KUKA KRL data list: CNC3.dat

&ACCESS RV
DEFDAT CNC3 Public
DECL GLOBAL FRAME gfCNCPoint3[30000]


gfCNCPoint3[1] = {X 137.7105, Y 20.4366, Z -3.8333, A 0.000, B 0.000, C 0.000 }
gfCNCPoint3[2] = {X 137.0001, Y 21.1821, Z -3.8333, A 0.000, B 0.000, C 0.000 }
gfCNCPoint3[3] = {X 136.1491, Y 21.7619, Z -3.8333, A 0.000, B 0.000, C 0.000 }
gfCNCPoint3[4] = {X 135.4282, Y 22.0767, Z -3.8333, A 0.000, B 0.000, C 0.000 }
gfCNCPoint3[5] = {X 134.6660, Y 22.2715, Z -3.8333, A 0.000, B 0.000, C 0.000 }
gfCNCPoint3[6] = {X 133.8824, Y 22.3414, Z -3.8333, A 0.000, B 0.000, C 0.000 }
gfCNCPoint3[7] = {X 133.2006, Y 22.3415, Z -3.8333, A 0.000, B 0.000, C 0.000 }
gfCNCPoint3[8] = {X 132.2486, Y 22.2478, Z -3.8333, A 0.000, B 0.000, C 0.000 }
gfCNCPoint3[9] = {X 131.3331, Y 21.9701, Z -3.8333, A 0.000, B 0.000, C 0.000 }
gfCNCPoint3[10] = {X 130.4895, Y 21.5191, Z -3.8333, A 0.000, B 0.000, C 0.000 }
gfCNCPoint3[11] = {X 129.7500, Y 20.9122, Z -3.8333, A 0.000, B 0.000, C 0.000 }
gfCNCPoint3[12] = {X 129.1431, Y 20.1727, Z -3.8333, A 0.000, B 0.000, C 0.000 }
gfCNCPoint3[13] = {X 128.6921, Y 19.3290, Z -3.8333, A 0.000, B 0.000, C 0.000 }
gfCNCPoint3[14] = {X 128.4144, Y 18.4136, Z -3.8333, A 0.000, B 0.000, C 0.000 }
gfCNCPoint3[15] = {X 128.3206, Y 17.4615, Z -3.8333, A 0.000, B 0.000, C 0.000 }
gfCNCPoint3[16] = {X 128.3206, Y 10.4835, Z -3.8333, A 0.000, B 0.000, C 0.000 }
gfCNCPoint3[17] = {X 128.3317, Y 10.1548, Z -3.8333, A 0.000, B 0.000, C 0.000 }
gfCNCPoint3[18] = {X 128.3649, Y 9.8276, Z -3.8333, A 0.000, B 0.000, C 0.000 }
gfCNCPoint3[19] = {X 128.6078, Y 8.8341, Z -3.8333, A 0.000, B 0.000, C 0.000 }
gfCNCPoint3[20] = {X 129.0525, Y 7.9131, Z -3.8333, A 0.000, B 0.000, C 0.000 }
gfCNCPoint3[21] = {X 129.6793, Y 7.1050, Z -3.8333, A 0.000, B 0.000, C 0.000 }
gfCNCPoint3[22] = {X 130.0256, Y 7.4373, Z -3.8333, A 0.000, B 0.000, C 0.000 }
gfCNCPoint3[23] = {X 130.6996, Y 6.8634, Z -3.8333, A 0.000, B 0.000, C 0.000 }
gfCNCPoint3[24] = {X 131.4749, Y 6.4361, Z -3.8333, A 0.000, B 0.000, C 0.000 }
gfCNCPoint3[25] = {X 132.3199, Y 6.1726, Z -3.8333, A 0.000, B 0.000, C 0.000 }
gfCNCPoint3[26] = {X 133.2007, Y 6.0835, Z -3.8333, A 0.000, B 0.000, C 0.000 }
gfCNCPoint3[27] = {X 133.8874, Y 6.0837, Z -3.8333, A 0.000, B 0.000, C 0.000 }
gfCNCPoint3[28] = {X 134.7189, Y 6.1717, Z -3.8333, A 0.000, B 0.000, C 0.000 }
gfCNCPoint3[29] = {X 135.5188, Y 6.4154, Z -3.8333, A 0.000, B 0.000, C 0.000 }
gfCNCPoint3[30] = {X 136.2581, Y 6.8060, Z -3.8333, A 0.000, B 0.000, C 0.000 }
gfCNCPoint3[31] = {X 136.9101, Y 7.3294, Z -3.8333, A 0.000, B 0.000, C 0.000 }
gfCNCPoint3[32] = {X 137.4514, Y 7.9667, Z -3.8333, A 0.000, B 0.000, C 0.000 }
gfCNCPoint3[33] = {X 155.0713, Y 7.9667, Z -3.8333, A 0.000, B 0.000, C 0.000 }
gfCNCPoint3[34] = {X 155.6191, Y 7.3231, Z -3.8333, A 0.000, B 0.000, C 0.000 }
gfCNCPoint3[35] = {X 156.2798, Y 6.7961, Z -3.8333, A 0.000, B 0.000, C 0.000 }
gfCNCPoint3[36] = {X 157.0291, Y 6.4051, Z -3.8333, A 0.000, B 0.000, C 0.000 }
gfCNCPoint3[37] = {X 157.8393, Y 6.1647, Z -3.8333, A 0.000, B 0.000, C 0.000 }
gfCNCPoint3[38] = {X 158.6806, Y 6.0835, Z -3.8333, A 0.000, B 0.000, C 0.000 }
gfCNCPoint3[39] = {X 159.3791, Y 6.0839, Z -3.8333, A 0.000, B 0.000, C 0.000 }
gfCNCPoint3[40] = {X 160.3488, Y 6.2050, Z -3.8333, A 0.000, B 0.000, C 0.000 }
gfCNCPoint3[41] = {X 161.2678, Y 6.5371, Z -3.8333, A 0.000, B 0.000, C 0.000 }
gfCNCPoint3[42] = {X 162.0908, Y 7.0639, Z -3.8333, A 0.000, B 0.000, C 0.000 }
gfCNCPoint3[43] = {X 162.7773, Y 7.7593, Z -3.8333, A 0.000, B 0.000, C 0.000 }
gfCNCPoint3[44] = {X 163.2934, Y 8.5891, Z -3.8333, A 0.000, B 0.000, C 0.000 }
gfCNCPoint3[45] = {X 163.6136, Y 9.5124, Z -3.8333, A 0.000, B 0.000, C 0.000 }
gfCNCPoint3[46] = {X 163.7221, Y 10.4835, Z -3.8333, A 0.000, B 0.000, C 0.000 }
gfCNCPoint3[47] = {X 163.7221, Y 17.4615, Z -3.8333, A 0.000, B 0.000, C 0.000 }
gfCNCPoint3[48] = {X 163.6118, Y 18.4406, Z -3.8333, A 0.000, B 0.000, C 0.000 }
gfCNCPoint3[49] = {X 163.2863, Y 19.3706, Z -3.8333, A 0.000, B 0.000, C 0.000 }
gfCNCPoint3[50] = {X 162.7621, Y 20.2049, Z -3.8333, A 0.000, B 0.000, C 0.000 }
gfCNCPoint3[51] = {X 162.0654, Y 20.9016, Z -3.8333, A 0.000, B 0.000, C 0.000 }
gfCNCPoint3[52] = {X 161.2312, Y 21.4258, Z -3.8333, A 0.000, B 0.000, C 0.000 }
gfCNCPoint3[53] = {X 160.3012, Y 21.7512, Z -3.8333, A 0.000, B 0.000, C 0.000 }
gfCNCPoint3[54] = {X 159.3221, Y 21.8615, Z -3.8333, A 0.000, B 0.000, C 0.000 }
gfCNCPoint3[55] = {X 158.6788, Y 21.8615, Z -3.8333, A 0.000, B 0.000, C 0.000 }
gfCNCPoint3[56] = {X 157.8334, Y 21.7764, Z -3.8333, A 0.000, B 0.000, C 0.000 }
gfCNCPoint3[57] = {X 157.0197, Y 21.5317, Z -3.8333, A 0.000, B 0.000, C 0.000 }
gfCNCPoint3[58] = {X 156.2677, Y 21.1363, Z -3.8333, A 0.000, B 0.000, C 0.000 }
gfCNCPoint3[59] = {X 155.6048, Y 20.6048, Z -3.8333, A 0.000, B 0.000, C 0.000 }
gfCNCPoint3[60] = {X 155.0554, Y 19.9566, Z -3.8333, A 0.000, B 0.000, C 0.000 }
gfCNCPoint3[61] = {X 152.3562, Y 19.9578, Z -3.8333, A 0.000, B 0.000, C 0.000 }
gfCNCPoint3[62] = {X 152.3548, Y 40.8428, Z -3.8333, A 0.000, B 0.000, C 0.000 }
gfCNCPoint3[63] = {X 152.8075, Y 41.3308, Z -3.8333, A 0.000, B 0.000, C 0.000 }
gfCNCPoint3[64] = {X 152.8997, Y 41.4410, Z -3.8333, A 0.000, B 0.000, C 0.000 }
gfCNCPoint3[65] = {X 153.4341, Y 42.2814, Z -3.8333, A 0.000, B 0.000, C 0.000 }
gfCNCPoint3[66] = {X 153.7674, Y 43.2198, Z -3.8333, A 0.000, B 0.000, C 0.000 }
gfCNCPoint3[67] = {X 153.8831, Y 44.2089, Z -3.8333, A 0.000, B 0.000, C 0.000 }
gfCNCPoint3[68] = {X 153.8829, Y 45.0423, Z -3.8333, A 0.000, B 0.000, C 0.000 }
gfCNCPoint3[69] = {X 153.7646, Y 46.0144, Z -3.8333, A 0.000, B 0.000, C 0.000 }
gfCNCPoint3[70] = {X 153.4342, Y 46.9363, Z -3.8333, A 0.000, B 0.000, C 0.000 }
gfCNCPoint3[71] = {X 152.9080, Y 47.7622, Z -3.8333, A 0.000, B 0.000, C 0.000 }
gfCNCPoint3[72] = {X 152.2123, Y 48.4513, Z -3.8333, A 0.000, B 0.000, C 0.000 }
gfCNCPoint3[73] = {X 151.3813, Y 48.9695, Z -3.8333, A 0.000, B 0.000, C 0.000 }
gfCNCPoint3[74] = {X 150.4563, Y 49.2910, Z -3.8333, A 0.000, B 0.000, C 0.000 }
gfCNCPoint3[75] = {X 149.4831, Y 49.4000, Z -3.8333, A 0.000, B 0.000, C 0.000 }
gfCNCPoint3[76] = {X 143.0396, Y 49.4000, Z -3.8333, A 0.000, B 0.000, C 0.000 }
gfCNCPoint3[77] = {X 142.0605, Y 49.2897, Z -3.8333, A 0.000, B 0.000, C 0.000 }
gfCNCPoint3[78] = {X 141.1305, Y 48.9643, Z -3.8333, A 0.000, B 0.000, C 0.000 }
gfCNCPoint3[79] = {X 140.2963, Y 48.4400, Z -3.8333, A 0.000, B 0.000, C 0.000 }
gfCNCPoint3[80] = {X 139.5996, Y 47.7433, Z -3.8333, A 0.000, B 0.000, C 0.000 }
gfCNCPoint3[81] = {X 139.0754, Y 46.9091, Z -3.8333, A 0.000, B 0.000, C 0.000 }
gfCNCPoint3[82] = {X 138.7499, Y 45.9791, Z -3.8333, A 0.000, B 0.000, C 0.000 }
gfCNCPoint3[83] = {X 138.6396, Y 45.0000, Z -3.8333, A 0.000, B 0.000, C 0.000 }
gfCNCPoint3[84] = {X 138.6400, Y 44.1483, Z -3.8333, A 0.000, B 0.000, C 0.000 }
gfCNCPoint3[85] = {X 138.7505, Y 43.2275, Z -3.8333, A 0.000, B 0.000, C 0.000 }
gfCNCPoint3[86] = {X 139.0514, Y 42.3503, Z -3.8333, A 0.000, B 0.000, C 0.000 }
gfCNCPoint3[87] = {X 139.5295, Y 41.5556, Z -3.8333, A 0.000, B 0.000, C 0.000 }
gfCNCPoint3[88] = {X 140.1636, Y 40.8789, Z -3.8333, A 0.000, B 0.000, C 0.000 }
gfCNCPoint3[89] = {X 140.1636, Y 19.9572, Z -3.8333, A 0.000, B 0.000, C 0.000 }
gfCNCPoint3[90] = {X 137.4665, Y 19.9566, Z -3.8333, A 0.000, B 0.000, C 0.000 }
gfCNCPoint3[91] = {X 136.9188, Y 20.6072, Z -3.8333, A 0.000, B 0.000, C 0.000 }
gfCNCPoint3[92] = {X 136.2562, Y 21.1403, Z -3.8333, A 0.000, B 0.000, C 0.000 }
gfCNCPoint3[93] = {X 135.5034, Y 21.5359, Z -3.8333, A 0.000, B 0.000, C 0.000 }
gfCNCPoint3[94] = {X 134.6886, Y 21.7794, Z -3.8333, A 0.000, B 0.000, C 0.000 }
gfCNCPoint3[95] = {X 133.8422, Y 21.8615, Z -3.8333, A 0.000, B 0.000, C 0.000 }
gfCNCPoint3[96] = {X 133.2006, Y 21.8615, Z -3.8333, A 0.000, B 0.000, C 0.000 }
gfCNCPoint3[97] = {X 132.2215, Y 21.7512, Z -3.8333, A 0.000, B 0.000, C 0.000 }
gfCNCPoint3[98] = {X 131.2916, Y 21.4258, Z -3.8333, A 0.000, B 0.000, C 0.000 }
gfCNCPoint3[99] = {X 130.4573, Y 20.9016, Z -3.8333, A 0.000, B 0.000, C 0.000 }
gfCNCPoint3[100] = {X 129.7606, Y 20.2049, Z -3.8333, A 0.000, B 0.000, C 0.000 }
gfCNCPoint3[101] = {X 129.2364, Y 19.3706, Z -3.8333, A 0.000, B 0.000, C 0.000 }
gfCNCPoint3[102] = {X 128.9110, Y 18.4406, Z -3.8333, A 0.000, B 0.000, C 0.000 }
gfCNCPoint3[103] = {X 128.8006, Y 17.4615, Z -3.8333, A 0.000, B 0.000, C 0.000 }
gfCNCPoint3[104] = {X 128.8006, Y 10.4835, Z -3.8333, A 0.000, B 0.000, C 0.000 }
gfCNCPoint3[105] = {X 128.8808, Y 9.6475, Z -3.8333, A 0.000, B 0.000, C 0.000 }
gfCNCPoint3[106] = {X 129.1184, Y 8.8419, Z -3.8333, A 0.000, B 0.000, C 0.000 }
gfCNCPoint3[107] = {X 129.5047, Y 8.0961, Z -3.8333, A 0.000, B 0.000, C 0.000 }
gfCNCPoint3[108] = {X 130.0256, Y 7.4373, Z -3.8333, A 0.000, B 0.000, C 0.000 }
gfCNCPoint3[109] = {X 129.6793, Y 7.1050, Z -3.8333, A 0.000, B 0.000, C 0.000 }
gfCNCPoint3[110] = {X 102.4337, Y 7.1050, Z -3.8333, A 0.000, B 0.000, C 0.000 }
gfCNCPoint3[111] = {X 102.4337, Y 11.9050, Z -3.8333, A 0.000, B 0.000, C 0.000 }
gfCNCPoint3[112] = {X 101.3242, Y 11.9050, Z -3.8333, A 0.000, B 0.000, C 0.000 }
gfCNCPoint3[113] = {X 101.3283, Y 12.0459, Z -3.8333, A 0.000, B 0.000, C 0.000 }
gfCNCPoint3[114] = {X 101.3297, Y 12.1868, Z -3.8333, A 0.000, B 0.000, C 0.000 }
gfCNCPoint3[115] = {X 101.3293, Y 13.0462, Z -3.8333, A 0.000, B 0.000, C 0.000 }
gfCNCPoint3[116] = {X 101.2274, Y 14.1939, Z -3.8333, A 0.000, B 0.000, C 0.000 }
gfCNCPoint3[117] = {X 100.9457, Y 15.3111, Z -3.8333, A 0.000, B 0.000, C 0.000 }
gfCNCPoint3[118] = {X 101.0393, Y 15.5442, Z -3.8333, A 0.000, B 0.000, C 0.000 }
gfCNCPoint3[119] = {X 101.8684, Y 17.5994, Z -3.8333, A 0.000, B 0.000, C 0.000 }
gfCNCPoint3[120] = {X 102.8003, Y 15.2755, Z -3.8333, A 0.000, B 0.000, C 0.000 }
gfCNCPoint3[121] = {X 102.5264, Y 14.1695, Z -3.8333, A 0.000, B 0.000, C 0.000 }
gfCNCPoint3[122] = {X 102.4285, Y 13.0344, Z -3.8333, A 0.000, B 0.000, C 0.000 }
gfCNCPoint3[123] = {X 102.4283, Y 12.1868, Z -3.8333, A 0.000, B 0.000, C 0.000 }
gfCNCPoint3[124] = {X 102.4296, Y 12.0459, Z -3.8333, A 0.000, B 0.000, C 0.000 }
gfCNCPoint3[125] = {X 102.4337, Y 11.9050, Z -3.8333, A 0.000, B 0.000, C 0.000 }
gfCNCPoint3[126] = {X 102.4337, Y 9.5050, Z -3.8333, A 0.000, B 0.000, C 0.000 }
gfCNCPoint3[127] = {X 98.1267, Y 9.5050, Z -3.8333, A 0.000, B 0.000, C 0.000 }
gfCNCPoint3[128] = {X 98.5429, Y 10.2829, Z -3.8333, A 0.000, B 0.000, C 0.000 }
gfCNCPoint3[129] = {X 98.8123, Y 11.1230, Z -3.8333, A 0.000, B 0.000, C 0.000 }
gfCNCPoint3[130] = {X 98.9260, Y 11.9979, Z -3.8333, A 0.000, B 0.000, C 0.000 }
gfCNCPoint3[131] = {X 98.9288, Y 12.0923, Z -3.8333, A 0.000, B 0.000, C 0.000 }
gfCNCPoint3[132] = {X 98.9297, Y 12.1868, Z -3.8333, A 0.000, B 0.000, C 0.000 }
gfCNCPoint3[133] = {X 98.9294, Y 13.0237, Z -3.8333, A 0.000, B 0.000, C 0.000 }
gfCNCPoint3[134] = {X 98.8589, Y 13.8059, Z -3.8333, A 0.000, B 0.000, C 0.000 }
gfCNCPoint3[135] = {X 98.6639, Y 14.5666, Z -3.8333, A 0.000, B 0.000, C 0.000 }
gfCNCPoint3[136] = {X 98.3493, Y 15.2862, Z -3.8333, A 0.000, B 0.000, C 0.000 }
gfCNCPoint3[137] = {X 98.8129, Y 16.4405, Z -3.8333, A 0.000, B 0.000, C 0.000 }
gfCNCPoint3[138] = {X 101.8752, Y 24.0312, Z -3.8333, A 0.000, B 0.000, C 0.000 }
gfCNCPoint3[139] = {X 105.3933, Y 15.2574, Z -3.8333, A 0.000, B 0.000, C 0.000 }
gfCNCPoint3[140] = {X 105.0870, Y 14.5458, Z -3.8333, A 0.000, B 0.000, C 0.000 }
gfCNCPoint3[141] = {X 104.8971, Y 13.7947, Z -3.8333, A 0.000, B 0.000, C 0.000 }
gfCNCPoint3[142] = {X 104.8285, Y 13.0231, Z -3.8333, A 0.000, B 0.000, C 0.000 }
gfCNCPoint3[143] = {X 104.8283, Y 12.1868, Z -3.8333, A 0.000, B 0.000, C 0.000 }
gfCNCPoint3[144] = {X 104.8292, Y 12.0923, Z -3.8333, A 0.000, B 0.000, C 0.000 }
gfCNCPoint3[145] = {X 104.8319, Y 11.9979, Z -3.8333, A 0.000, B 0.000, C 0.000 }
gfCNCPoint3[146] = {X 104.9456, Y 11.1230, Z -3.8333, A 0.000, B 0.000, C 0.000 }
gfCNCPoint3[147] = {X 105.2150, Y 10.2829, Z -3.8333, A 0.000, B 0.000, C 0.000 }
gfCNCPoint3[148] = {X 105.6312, Y 9.5050, Z -3.8333, A 0.000, B 0.000, C 0.000 }
gfCNCPoint3[149] = {X 102.4337, Y 9.5050, Z -3.8333, A 0.000, B 0.000, C 0.000 }
gfCNCPoint3[150] = {X 102.4337, Y 7.1050, Z -3.8333, A 0.000, B 0.000, C 0.000 }
gfCNCPoint3[151] = {X 64.8350, Y 7.1050, Z -3.8333, A 0.000, B 0.000, C 0.000 }
gfCNCPoint3[152] = {X 65.5946, Y 8.0242, Z -3.8333, A 0.000, B 0.000, C 0.000 }
gfCNCPoint3[153] = {X 66.1941, Y 9.0550, Z -3.8333, A 0.000, B 0.000, C 0.000 }
gfCNCPoint3[154] = {X 66.6172, Y 10.1699, Z -3.8333, A 0.000, B 0.000, C 0.000 }
gfCNCPoint3[155] = {X 66.8305, Y 11.1683, Z -3.8333, A 0.000, B 0.000, C 0.000 }
gfCNCPoint3[156] = {X 66.9021, Y 12.1868, Z -3.8333, A 0.000, B 0.000, C 0.000 }
gfCNCPoint3[157] = {X 66.9018, Y 13.0462, Z -3.8333, A 0.000, B 0.000, C 0.000 }
gfCNCPoint3[158] = {X 66.7772, Y 14.3210, Z -3.8333, A 0.000, B 0.000, C 0.000 }
gfCNCPoint3[159] = {X 66.4310, Y 15.5543, Z -3.8333, A 0.000, B 0.000, C 0.000 }
gfCNCPoint3[160] = {X 74.9112, Y 38.2391, Z -3.8333, A 0.000, B 0.000, C 0.000 }
gfCNCPoint3[161] = {X 75.8036, Y 38.9739, Z -3.8333, A 0.000, B 0.000, C 0.000 }
gfCNCPoint3[162] = {X 76.5684, Y 39.8407, Z -3.8333, A 0.000, B 0.000, C 0.000 }
gfCNCPoint3[163] = {X 77.1864, Y 40.8176, Z -3.8333, A 0.000, B 0.000, C 0.000 }
gfCNCPoint3[164] = {X 77.6419, Y 41.8800, Z -3.8333, A 0.000, B 0.000, C 0.000 }
gfCNCPoint3[165] = {X 77.9236, Y 43.0011, Z -3.8333, A 0.000, B 0.000, C 0.000 }
gfCNCPoint3[166] = {X 78.0243, Y 44.1527, Z -3.8333, A 0.000, B 0.000, C 0.000 }
gfCNCPoint3[167] = {X 78.0245, Y 45.0000, Z -3.8333, A 0.000, B 0.000, C 0.000 }
gfCNCPoint3[168] = {X 77.9139, Y 46.2642, Z -3.8333, A 0.000, B 0.000, C 0.000 }
gfCNCPoint3[169] = {X 77.5854, Y 47.4899, Z -3.8333, A 0.000, B 0.000, C 0.000 }
gfCNCPoint3[170] = {X 77.0491, Y 48.6400, Z -3.8333, A 0.000, B 0.000, C 0.000 }
gfCNCPoint3[171] = {X 76.3213, Y 49.6795, Z -3.8333, A 0.000, B 0.000, C 0.000 }
gfCNCPoint3[172] = {X 75.4240, Y 50.5768, Z -3.8333, A 0.000, B 0.000, C 0.000 }
gfCNCPoint3[173] = {X 74.3845, Y 51.3047, Z -3.8333, A 0.000, B 0.000, C 0.000 }
gfCNCPoint3[174] = {X 73.2344, Y 51.8410, Z -3.8333, A 0.000, B 0.000, C 0.000 }
gfCNCPoint3[175] = {X 72.0086, Y 52.1694, Z -3.8333, A 0.000, B 0.000, C 0.000 }
gfCNCPoint3[176] = {X 70.7445, Y 52.2800, Z -3.8333, A 0.000, B 0.000, C 0.000 }
gfCNCPoint3[177] = {X 64.1851, Y 52.2800, Z -3.8333, A 0.000, B 0.000, C 0.000 }
gfCNCPoint3[178] = {X 62.9397, Y 52.1727, Z -3.8333, A 0.000, B 0.000, C 0.000 }
gfCNCPoint3[179] = {X 61.7311, Y 51.8539, Z -3.8333, A 0.000, B 0.000, C 0.000 }
gfCNCPoint3[180] = {X 60.5947, Y 51.3330, Z -3.8333, A 0.000, B 0.000, C 0.000 }
gfCNCPoint3[181] = {X 59.5643, Y 50.6255, Z -3.8333, A 0.000, B 0.000, C 0.000 }
gfCNCPoint3[182] = {X 58.6700, Y 49.7521, Z -3.8333, A 0.000, B 0.000, C 0.000 }
gfCNCPoint3[183] = {X 57.9384, Y 48.7385, Z -3.8333, A 0.000, B 0.000, C 0.000 }
gfCNCPoint3[184] = {X 57.3706, Y 47.5614, Z -3.8333, A 0.000, B 0.000, C 0.000 }
gfCNCPoint3[185] = {X 57.0224, Y 46.3017, Z -3.8333, A 0.000, B 0.000, C 0.000 }
gfCNCPoint3[186] = {X 56.9051, Y 45.0000, Z -3.8333, A 0.000, B 0.000, C 0.000 }
gfCNCPoint3[187] = {X 56.9051, Y 44.2047, Z -3.8333, A 0.000, B 0.000, C 0.000 }
gfCNCPoint3[188] = {X 56.9286, Y 43.6251, Z -3.8333, A 0.000, B 0.000, C 0.000 }
gfCNCPoint3[189] = {X 56.9981, Y 43.0492, Z -3.8333, A 0.000, B 0.000, C 0.000 }
gfCNCPoint3[190] = {X 54.7600, Y 43.0492, Z -3.8333, A 0.000, B 0.000, C 0.000 }
gfCNCPoint3[191] = {X 54.8275, Y 43.6012, Z -3.8333, A 0.000, B 0.000, C 0.000 }
gfCNCPoint3[192] = {X 54.8527, Y 44.1567, Z -3.8333, A 0.000, B 0.000, C 0.000 }
gfCNCPoint3[193] = {X 54.8529, Y 45.0000, Z -3.8333, A 0.000, B 0.000, C 0.000 }
gfCNCPoint3[194] = {X 54.7356, Y 46.3017, Z -3.8333, A 0.000, B 0.000, C 0.000 }
gfCNCPoint3[195] = {X 54.3875, Y 47.5614, Z -3.8333, A 0.000, B 0.000, C 0.000 }
gfCNCPoint3[196] = {X 53.8197, Y 48.7385, Z -3.8333, A 0.000, B 0.000, C 0.000 }
gfCNCPoint3[197] = {X 53.0880, Y 49.7521, Z -3.8333, A 0.000, B 0.000, C 0.000 }
gfCNCPoint3[198] = {X 52.1938, Y 50.6255, Z -3.8333, A 0.000, B 0.000, C 0.000 }
gfCNCPoint3[199] = {X 51.1633, Y 51.3330, Z -3.8333, A 0.000, B 0.000, C 0.000 }
gfCNCPoint3[200] = {X 50.0270, Y 51.8539, Z -3.8333, A 0.000, B 0.000, C 0.000 }
gfCNCPoint3[201] = {X 48.8183, Y 52.1727, Z -3.8333, A 0.000, B 0.000, C 0.000 }
gfCNCPoint3[202] = {X 47.5729, Y 52.2800, Z -3.8333, A 0.000, B 0.000, C 0.000 }
gfCNCPoint3[203] = {X 40.6393, Y 52.2800, Z -3.8333, A 0.000, B 0.000, C 0.000 }
gfCNCPoint3[204] = {X 39.4476, Y 52.1818, Z -3.8333, A 0.000, B 0.000, C 0.000 }
gfCNCPoint3[205] = {X 38.2881, Y 51.8899, Z -3.8333, A 0.000, B 0.000, C 0.000 }
gfCNCPoint3[206] = {X 37.1919, Y 51.4120, Z -3.8333, A 0.000, B 0.000, C 0.000 }
gfCNCPoint3[207] = {X 36.1888, Y 50.7612, Z -3.8333, A 0.000, B 0.000, C 0.000 }
gfCNCPoint3[208] = {X 35.3058, Y 49.9550, Z -3.8333, A 0.000, B 0.000, C 0.000 }
gfCNCPoint3[209] = {X 34.8234, Y 50.4196, Z -3.8333, A 0.000, B 0.000, C 0.000 }
gfCNCPoint3[210] = {X 34.3150, Y 50.8555, Z -3.8333, A 0.000, B 0.000, C 0.000 }
gfCNCPoint3[211] = {X 33.7743, Y 51.2926, Z -3.8333, A 0.000, B 0.000, C 0.000 }
gfCNCPoint3[212] = {X 32.5161, Y 52.1774, Z -3.8333, A 0.000, B 0.000, C 0.000 }
gfCNCPoint3[213] = {X 31.1520, Y 52.8883, Z -3.8333, A 0.000, B 0.000, C 0.000 }
gfCNCPoint3[214] = {X 29.7059, Y 53.4126, Z -3.8333, A 0.000, B 0.000, C 0.000 }
gfCNCPoint3[215] = {X 28.2032, Y 53.7412, Z -3.8333, A 0.000, B 0.000, C 0.000 }
gfCNCPoint3[216] = {X 26.6703, Y 53.8684, Z -3.8333, A 0.000, B 0.000, C 0.000 }
gfCNCPoint3[217] = {X 24.3221, Y 54.9119, Z -3.8333, A 0.000, B 0.000, C 0.000 }
gfCNCPoint3[218] = {X 21.9059, Y 55.7866, Z -3.8333, A 0.000, B 0.000, C 0.000 }
gfCNCPoint3[219] = {X 19.5313, Y 56.4616, Z -3.8333, A 0.000, B 0.000, C 0.000 }
gfCNCPoint3[220] = {X 17.1094, Y 56.9400, Z -3.8333, A 0.000, B 0.000, C 0.000 }
gfCNCPoint3[221] = {X 14.6565, Y 57.2186, Z -3.8333, A 0.000, B 0.000, C 0.000 }
gfCNCPoint3[222] = {X 12.1890, Y 57.2954, Z -3.8333, A 0.000, B 0.000, C 0.000 }
gfCNCPoint3[223] = {X 9.7235, Y 57.1699, Z -3.8333, A 0.000, B 0.000, C 0.000 }
gfCNCPoint3[224] = {X 8.4096, Y 57.0199, Z -3.8333, A 0.000, B 0.000, C 0.000 }
gfCNCPoint3[225] = {X 7.1035, Y 56.8124, Z -3.8333, A 0.000, B 0.000, C 0.000 }
gfCNCPoint3[226] = {X 7.1035, Y 92.8950, Z -3.8333, A 0.000, B 0.000, C 0.000 }
gfCNCPoint3[227] = {X 116.2647, Y 92.8950, Z -3.8333, A 0.000, B 0.000, C 0.000 }
gfCNCPoint3[228] = {X 116.9737, Y 91.6538, Z -3.8333, A 0.000, B 0.000, C 0.000 }
gfCNCPoint3[229] = {X 117.8578, Y 90.5306, Z -3.8333, A 0.000, B 0.000, C 0.000 }
gfCNCPoint3[230] = {X 118.8976, Y 89.5497, Z -3.8333, A 0.000, B 0.000, C 0.000 }
gfCNCPoint3[231] = {X 120.0706, Y 88.7328, Z -3.8333, A 0.000, B 0.000, C 0.000 }
gfCNCPoint3[232] = {X 121.3510, Y 88.0974, Z -3.8333, A 0.000, B 0.000, C 0.000 }
gfCNCPoint3[233] = {X 122.7111, Y 87.6576, Z -3.8333, A 0.000, B 0.000, C 0.000 }
gfCNCPoint3[234] = {X 124.1211, Y 87.4228, Z -3.8333, A 0.000, B 0.000, C 0.000 }
gfCNCPoint3[235] = {X 124.5371, Y 87.3611, Z -3.8333, A 0.000, B 0.000, C 0.000 }
gfCNCPoint3[236] = {X 125.0284, Y 86.8587, Z -3.8333, A 0.000, B 0.000, C 0.000 }
gfCNCPoint3[237] = {X 125.5056, Y 86.3431, Z -3.8333, A 0.000, B 0.000, C 0.000 }
gfCNCPoint3[238] = {X 149.6586, Y 59.8197, Z -3.8333, A 0.000, B 0.000, C 0.000 }
gfCNCPoint3[239] = {X 149.6295, Y 59.4068, Z -3.8333, A 0.000, B 0.000, C 0.000 }
gfCNCPoint3[240] = {X 149.6181, Y 58.9930, Z -3.8333, A 0.000, B 0.000, C 0.000 }
gfCNCPoint3[241] = {X 149.6180, Y 58.0000, Z -3.8333, A 0.000, B 0.000, C 0.000 }
gfCNCPoint3[242] = {X 149.6915, Y 56.8093, Z -3.8333, A 0.000, B 0.000, C 0.000 }
gfCNCPoint3[243] = {X 149.9109, Y 55.6367, Z -3.8333, A 0.000, B 0.000, C 0.000 }
gfCNCPoint3[244] = {X 150.2729, Y 54.5000, Z -3.8333, A 0.000, B 0.000, C 0.000 }
gfCNCPoint3[245] = {X 150.7719, Y 53.4164, Z -3.8333, A 0.000, B 0.000, C 0.000 }
gfCNCPoint3[246] = {X 151.5117, Y 52.2488, Z -3.8333, A 0.000, B 0.000, C 0.000 }
gfCNCPoint3[247] = {X 152.4103, Y 51.1984, Z -3.8333, A 0.000, B 0.000, C 0.000 }
gfCNCPoint3[248] = {X 153.4493, Y 50.2867, Z -3.8333, A 0.000, B 0.000, C 0.000 }
gfCNCPoint3[249] = {X 154.6075, Y 49.5323, Z -3.8333, A 0.000, B 0.000, C 0.000 }
gfCNCPoint3[250] = {X 155.8614, Y 48.9505, Z -3.8333, A 0.000, B 0.000, C 0.000 }
gfCNCPoint3[251] = {X 157.1854, Y 48.5533, Z -3.8333, A 0.000, B 0.000, C 0.000 }
gfCNCPoint3[252] = {X 158.2353, Y 48.3785, Z -3.8333, A 0.000, B 0.000, C 0.000 }
gfCNCPoint3[253] = {X 159.2980, Y 48.3200, Z -3.8333, A 0.000, B 0.000, C 0.000 }
gfCNCPoint3[254] = {X 176.3103, Y 48.3200, Z -3.8333, A 0.000, B 0.000, C 0.000 }
gfCNCPoint3[255] = {X 175.1960, Y 47.6608, Z -3.8333, A 0.000, B 0.000, C 0.000 }
gfCNCPoint3[256] = {X 174.1332, Y 46.9214, Z -3.8333, A 0.000, B 0.000, C 0.000 }
gfCNCPoint3[257] = {X 172.7673, Y 45.7588, Z -3.8333, A 0.000, B 0.000, C 0.000 }
gfCNCPoint3[258] = {X 171.5638, Y 44.4288, Z -3.8333, A 0.000, B 0.000, C 0.000 }
gfCNCPoint3[259] = {X 170.6258, Y 43.0901, Z -3.8333, A 0.000, B 0.000, C 0.000 }
gfCNCPoint3[260] = {X 169.8528, Y 41.6499, Z -3.8333, A 0.000, B 0.000, C 0.000 }
gfCNCPoint3[261] = {X 169.2555, Y 40.1283, Z -3.8333, A 0.000, B 0.000, C 0.000 }
gfCNCPoint3[262] = {X 168.8424, Y 38.5468, Z -3.8333, A 0.000, B 0.000, C 0.000 }
gfCNCPoint3[263] = {X 168.6193, Y 36.9275, Z -3.8333, A 0.000, B 0.000, C 0.000 }
gfCNCPoint3[264] = {X 168.5331, Y 35.0259, Z -3.8333, A 0.000, B 0.000, C 0.000 }
gfCNCPoint3[265] = {X 168.6853, Y 33.1284, Z -3.8333, A 0.000, B 0.000, C 0.000 }
gfCNCPoint3[266] = {X 169.0736, Y 31.2648, Z -3.8333, A 0.000, B 0.000, C 0.000 }
gfCNCPoint3[267] = {X 169.6918, Y 29.4644, Z -3.8333, A 0.000, B 0.000, C 0.000 }
gfCNCPoint3[268] = {X 170.2638, Y 28.2677, Z -3.8333, A 0.000, B 0.000, C 0.000 }
gfCNCPoint3[269] = {X 170.9708, Y 27.1454, Z -3.8333, A 0.000, B 0.000, C 0.000 }
gfCNCPoint3[270] = {X 171.8031, Y 26.1126, Z -3.8333, A 0.000, B 0.000, C 0.000 }
gfCNCPoint3[271] = {X 172.7495, Y 25.1833, Z -3.8333, A 0.000, B 0.000, C 0.000 }
gfCNCPoint3[272] = {X 173.7973, Y 24.3700, Z -3.8333, A 0.000, B 0.000, C 0.000 }
gfCNCPoint3[273] = {X 173.0271, Y 23.7518, Z -3.8333, A 0.000, B 0.000, C 0.000 }
gfCNCPoint3[274] = {X 172.3971, Y 22.9912, Z -3.8333, A 0.000, B 0.000, C 0.000 }
gfCNCPoint3[275] = {X 171.9332, Y 22.1192, Z -3.8333, A 0.000, B 0.000, C 0.000 }
gfCNCPoint3[276] = {X 169.3220, Y 15.7237, Z -3.8333, A 0.000, B 0.000, C 0.000 }
gfCNCPoint3[277] = {X 169.1088, Y 15.0753, Z -3.8333, A 0.000, B 0.000, C 0.000 }
gfCNCPoint3[278] = {X 168.9882, Y 14.4035, Z -3.8333, A 0.000, B 0.000, C 0.000 }
gfCNCPoint3[279] = {X 168.9599, Y 13.8791, Z -3.8333, A 0.000, B 0.000, C 0.000 }
gfCNCPoint3[280] = {X 168.9882, Y 13.3548, Z -3.8333, A 0.000, B 0.000, C 0.000 }
gfCNCPoint3[281] = {X 169.1590, Y 12.4995, Z -3.8333, A 0.000, B 0.000, C 0.000 }
gfCNCPoint3[282] = {X 169.4794, Y 11.6883, Z -3.8333, A 0.000, B 0.000, C 0.000 }
gfCNCPoint3[283] = {X 169.9390, Y 10.9470, Z -3.8333, A 0.000, B 0.000, C 0.000 }
gfCNCPoint3[284] = {X 170.6135, Y 10.2179, Z -3.8333, A 0.000, B 0.000, C 0.000 }
gfCNCPoint3[285] = {X 171.4217, Y 9.6404, Z -3.8333, A 0.000, B 0.000, C 0.000 }
gfCNCPoint3[286] = {X 172.0576, Y 9.2779, Z -3.8333, A 0.000, B 0.000, C 0.000 }
gfCNCPoint3[287] = {X 172.9937, Y 8.8768, Z -3.8333, A 0.000, B 0.000, C 0.000 }
gfCNCPoint3[288] = {X 173.9927, Y 8.6787, Z -3.8333, A 0.000, B 0.000, C 0.000 }
gfCNCPoint3[289] = {X 175.0111, Y 8.6923, Z -3.8333, A 0.000, B 0.000, C 0.000 }
gfCNCPoint3[290] = {X 176.0044, Y 8.9170, Z -3.8333, A 0.000, B 0.000, C 0.000 }
gfCNCPoint3[291] = {X 177.7783, Y 8.1690, Z -3.8333, A 0.000, B 0.000, C 0.000 }
gfCNCPoint3[292] = {X 179.6059, Y 7.5638, Z -3.8333, A 0.000, B 0.000, C 0.000 }
gfCNCPoint3[293] = {X 181.4756, Y 7.1050, Z -3.8333, A 0.000, B 0.000, C 0.000 }
gfCNCPoint3[294] = {X 168.0205, Y 7.1050, Z -3.8333, A 0.000, B 0.000, C 0.000 }
gfCNCPoint3[295] = {X 168.0205, Y 4.7050, Z -3.8333, A 0.000, B 0.000, C 0.000 }
gfCNCPoint3[296] = {X 155.1590, Y 4.7050, Z -3.8333, A 0.000, B 0.000, C 0.000 }
gfCNCPoint3[297] = {X 155.1590, Y 7.1050, Z -3.8333, A 0.000, B 0.000, C 0.000 }
gfCNCPoint3[298] = {X 137.3637, Y 7.1050, Z -3.8333, A 0.000, B 0.000, C 0.000 }
gfCNCPoint3[299] = {X 137.5336, Y 7.2916, Z -3.8333, A 0.000, B 0.000, C 0.000 }
gfCNCPoint3[300] = {X 137.6937, Y 7.4867, Z -3.8333, A 0.000, B 0.000, C 0.000 }
gfCNCPoint3[301] = {X 154.8290, Y 7.4867, Z -3.8333, A 0.000, B 0.000, C 0.000 }
gfCNCPoint3[302] = {X 154.9891, Y 7.2916, Z -3.8333, A 0.000, B 0.000, C 0.000 }
gfCNCPoint3[303] = {X 155.1590, Y 7.1050, Z -3.8333, A 0.000, B 0.000, C 0.000 }
gfCNCPoint3[304] = {X 155.1590, Y 4.7050, Z -3.8333, A 0.000, B 0.000, C 0.000 }
gfCNCPoint3[305] = {X 42.6031, Y 4.7050, Z -3.8333, A 0.000, B 0.000, C 0.000 }
gfCNCPoint3[306] = {X 42.6031, Y 9.5050, Z -3.8333, A 0.000, B 0.000, C 0.000 }
gfCNCPoint3[307] = {X 36.0455, Y 9.5050, Z -3.8333, A 0.000, B 0.000, C 0.000 }
gfCNCPoint3[308] = {X 37.0557, Y 11.3888, Z -3.8333, A 0.000, B 0.000, C 0.000 }
gfCNCPoint3[309] = {X 37.8841, Y 13.3593, Z -3.8333, A 0.000, B 0.000, C 0.000 }
gfCNCPoint3[310] = {X 38.5465, Y 15.5412, Z -3.8333, A 0.000, B 0.000, C 0.000 }
gfCNCPoint3[311] = {X 39.0048, Y 17.7750, Z -3.8333, A 0.000, B 0.000, C 0.000 }
gfCNCPoint3[312] = {X 39.2551, Y 20.0415, Z -3.8333, A 0.000, B 0.000, C 0.000 }
gfCNCPoint3[313] = {X 39.2953, Y 22.3214, Z -3.8333, A 0.000, B 0.000, C 0.000 }
gfCNCPoint3[314] = {X 39.1250, Y 24.5953, Z -3.8333, A 0.000, B 0.000, C 0.000 }
gfCNCPoint3[315] = {X 42.5394, Y 15.4280, Z -3.8333, A 0.000, B 0.000, C 0.000 }
gfCNCPoint3[316] = {X 42.3081, Y 14.2497, Z -3.8333, A 0.000, B 0.000, C 0.000 }
gfCNCPoint3[317] = {X 42.2245, Y 13.0518, Z -3.8333, A 0.000, B 0.000, C 0.000 }
gfCNCPoint3[318] = {X 42.2242, Y 12.1868, Z -3.8333, A 0.000, B 0.000, C 0.000 }
gfCNCPoint3[319] = {X 42.3194, Y 10.8326, Z -3.8333, A 0.000, B 0.000, C 0.000 }
gfCNCPoint3[320] = {X 42.6031, Y 9.5050, Z -3.8333, A 0.000, B 0.000, C 0.000 }
gfCNCPoint3[321] = {X 42.6031, Y 7.1050, Z -3.8333, A 0.000, B 0.000, C 0.000 }
gfCNCPoint3[322] = {X 31.2110, Y 7.1050, Z -3.8333, A 0.000, B 0.000, C 0.000 }
gfCNCPoint3[323] = {X 32.2265, Y 8.2450, Z -3.8333, A 0.000, B 0.000, C 0.000 }
gfCNCPoint3[324] = {X 33.1533, Y 9.4582, Z -3.8333, A 0.000, B 0.000, C 0.000 }
gfCNCPoint3[325] = {X 33.9863, Y 10.7377, Z -3.8333, A 0.000, B 0.000, C 0.000 }
gfCNCPoint3[326] = {X 34.8870, Y 12.4168, Z -3.8333, A 0.000, B 0.000, C 0.000 }
gfCNCPoint3[327] = {X 35.6262, Y 14.1730, Z -3.8333, A 0.000, B 0.000, C 0.000 }
gfCNCPoint3[328] = {X 36.2226, Y 16.1409, Z -3.8333, A 0.000, B 0.000, C 0.000 }
gfCNCPoint3[329] = {X 36.6351, Y 18.1554, Z -3.8333, A 0.000, B 0.000, C 0.000 }
gfCNCPoint3[330] = {X 36.8603, Y 20.1993, Z -3.8333, A 0.000, B 0.000, C 0.000 }
gfCNCPoint3[331] = {X 36.8962, Y 22.2553, Z -3.8333, A 0.000, B 0.000, C 0.000 }
gfCNCPoint3[332] = {X 36.7425, Y 24.3058, Z -3.8333, A 0.000, B 0.000, C 0.000 }
gfCNCPoint3[333] = {X 36.5498, Y 25.5823, Z -3.8333, A 0.000, B 0.000, C 0.000 }
gfCNCPoint3[334] = {X 36.2834, Y 26.8455, Z -3.8333, A 0.000, B 0.000, C 0.000 }
gfCNCPoint3[335] = {X 35.8745, Y 28.3053, Z -3.8333, A 0.000, B 0.000, C 0.000 }
gfCNCPoint3[336] = {X 35.3504, Y 29.7277, Z -3.8333, A 0.000, B 0.000, C 0.000 }
gfCNCPoint3[337] = {X 34.7144, Y 31.1038, Z -3.8333, A 0.000, B 0.000, C 0.000 }
gfCNCPoint3[338] = {X 37.2846, Y 36.4132, Z -3.8333, A 0.000, B 0.000, C 0.000 }
gfCNCPoint3[339] = {X 41.3741, Y 25.4330, Z -3.8333, A 0.000, B 0.000, C 0.000 }
gfCNCPoint3[340] = {X 45.0743, Y 15.4981, Z -3.8333, A 0.000, B 0.000, C 0.000 }
gfCNCPoint3[341] = {X 44.7426, Y 14.2853, Z -3.8333, A 0.000, B 0.000, C 0.000 }
gfCNCPoint3[342] = {X 44.6244, Y 13.0334, Z -3.8333, A 0.000, B 0.000, C 0.000 }
gfCNCPoint3[343] = {X 44.6242, Y 12.1868, Z -3.8333, A 0.000, B 0.000, C 0.000 }
gfCNCPoint3[344] = {X 44.6958, Y 11.1683, Z -3.8333, A 0.000, B 0.000, C 0.000 }
gfCNCPoint3[345] = {X 44.9092, Y 10.1699, Z -3.8333, A 0.000, B 0.000, C 0.000 }
gfCNCPoint3[346] = {X 45.3323, Y 9.0550, Z -3.8333, A 0.000, B 0.000, C 0.000 }
gfCNCPoint3[347] = {X 45.9317, Y 8.0242, Z -3.8333, A 0.000, B 0.000, C 0.000 }
gfCNCPoint3[348] = {X 46.6914, Y 7.1050, Z -3.8333, A 0.000, B 0.000, C 0.000 }
gfCNCPoint3[349] = {X 42.6031, Y 7.1050, Z -3.8333, A 0.000, B 0.000, C 0.000 }
gfCNCPoint3[350] = {X 42.6031, Y 4.7050, Z -3.8333, A 0.000, B 0.000, C 0.000 }
gfCNCPoint3[351] = {X 23.8344, Y 4.7050, Z -3.8333, A 0.000, B 0.000, C 0.000 }
gfCNCPoint3[352] = {X 25.7632, Y 5.7852, Z -3.8333, A 0.000, B 0.000, C 0.000 }
gfCNCPoint3[353] = {X 27.5758, Y 7.0507, Z -3.8333, A 0.000, B 0.000, C 0.000 }
gfCNCPoint3[354] = {X 28.5589, Y 7.8750, Z -3.8333, A 0.000, B 0.000, C 0.000 }
gfCNCPoint3[355] = {X 29.4803, Y 8.7677, Z -3.8333, A 0.000, B 0.000, C 0.000 }
gfCNCPoint3[356] = {X 30.6887, Y 10.1631, Z -3.8333, A 0.000, B 0.000, C 0.000 }
gfCNCPoint3[357] = {X 31.7467, Y 11.6757, Z -3.8333, A 0.000, B 0.000, C 0.000 }
gfCNCPoint3[358] = {X 32.6431, Y 13.2893, Z -3.8333, A 0.000, B 0.000, C 0.000 }
gfCNCPoint3[359] = {X 33.3683, Y 14.9867, Z -3.8333, A 0.000, B 0.000, C 0.000 }
gfCNCPoint3[360] = {X 33.9180, Y 16.8175, Z -3.8333, A 0.000, B 0.000, C 0.000 }
gfCNCPoint3[361] = {X 34.2894, Y 18.6926, Z -3.8333, A 0.000, B 0.000, C 0.000 }
gfCNCPoint3[362] = {X 34.4791, Y 20.5946, Z -3.8333, A 0.000, B 0.000, C 0.000 }
gfCNCPoint3[363] = {X 34.4855, Y 22.5061, Z -3.8333, A 0.000, B 0.000, C 0.000 }
gfCNCPoint3[364] = {X 34.3083, Y 24.4094, Z -3.8333, A 0.000, B 0.000, C 0.000 }
gfCNCPoint3[365] = {X 33.9493, Y 26.2868, Z -3.8333, A 0.000, B 0.000, C 0.000 }
gfCNCPoint3[366] = {X 33.4657, Y 27.9387, Z -3.8333, A 0.000, B 0.000, C 0.000 }
gfCNCPoint3[367] = {X 32.8133, Y 29.5316, Z -3.8333, A 0.000, B 0.000, C 0.000 }
gfCNCPoint3[368] = {X 31.9991, Y 31.0481, Z -3.8333, A 0.000, B 0.000, C 0.000 }
gfCNCPoint3[369] = {X 32.1287, Y 31.2841, Z -3.8333, A 0.000, B 0.000, C 0.000 }
gfCNCPoint3[370] = {X 32.2513, Y 31.5237, Z -3.8333, A 0.000, B 0.000, C 0.000 }
gfCNCPoint3[371] = {X 35.3025, Y 37.8269, Z -3.8333, A 0.000, B 0.000, C 0.000 }
gfCNCPoint3[372] = {X 35.7263, Y 38.8573, Z -3.8333, A 0.000, B 0.000, C 0.000 }
gfCNCPoint3[373] = {X 36.0224, Y 39.9313, Z -3.8333, A 0.000, B 0.000, C 0.000 }
gfCNCPoint3[374] = {X 36.1865, Y 41.0332, Z -3.8333, A 0.000, B 0.000, C 0.000 }
gfCNCPoint3[375] = {X 36.2163, Y 42.1469, Z -3.8333, A 0.000, B 0.000, C 0.000 }
gfCNCPoint3[376] = {X 36.6304, Y 41.4261, Z -3.8333, A 0.000, B 0.000, C 0.000 }
gfCNCPoint3[377] = {X 37.1610, Y 40.7860, Z -3.8333, A 0.000, B 0.000, C 0.000 }
gfCNCPoint3[378] = {X 37.7924, Y 40.2452, Z -3.8333, A 0.000, B 0.000, C 0.000 }
gfCNCPoint3[379] = {X 38.5065, Y 39.8195, Z -3.8333, A 0.000, B 0.000, C 0.000 }
gfCNCPoint3[380] = {X 39.0451, Y 38.5339, Z -3.8333, A 0.000, B 0.000, C 0.000 }
gfCNCPoint3[381] = {X 39.5409, Y 37.2311, Z -3.8333, A 0.000, B 0.000, C 0.000 }
gfCNCPoint3[382] = {X 47.6703, Y 15.4045, Z -3.8333, A 0.000, B 0.000, C 0.000 }
gfCNCPoint3[383] = {X 47.3200, Y 14.6512, Z -3.8333, A 0.000, B 0.000, C 0.000 }
gfCNCPoint3[384] = {X 47.1026, Y 13.8493, Z -3.8333, A 0.000, B 0.000, C 0.000 }
gfCNCPoint3[385] = {X 47.0244, Y 13.0222, Z -3.8333, A 0.000, B 0.000, C 0.000 }
gfCNCPoint3[386] = {X 47.0242, Y 12.1868, Z -3.8333, A 0.000, B 0.000, C 0.000 }
gfCNCPoint3[387] = {X 47.1150, Y 11.2500, Z -3.8333, A 0.000, B 0.000, C 0.000 }
gfCNCPoint3[388] = {X 47.3839, Y 10.3480, Z -3.8333, A 0.000, B 0.000, C 0.000 }
gfCNCPoint3[389] = {X 47.8210, Y 9.5145, Z -3.8333, A 0.000, B 0.000, C 0.000 }
gfCNCPoint3[390] = {X 48.4099, Y 8.7803, Z -3.8333, A 0.000, B 0.000, C 0.000 }
gfCNCPoint3[391] = {X 49.1544, Y 8.1553, Z -3.8333, A 0.000, B 0.000, C 0.000 }
gfCNCPoint3[392] = {X 50.0081, Y 7.6903, Z -3.8333, A 0.000, B 0.000, C 0.000 }
gfCNCPoint3[393] = {X 50.9370, Y 7.4036, Z -3.8333, A 0.000, B 0.000, C 0.000 }
gfCNCPoint3[394] = {X 51.9042, Y 7.3068, Z -3.8333, A 0.000, B 0.000, C 0.000 }
gfCNCPoint3[395] = {X 59.6221, Y 7.3068, Z -3.8333, A 0.000, B 0.000, C 0.000 }
gfCNCPoint3[396] = {X 60.5894, Y 7.4036, Z -3.8333, A 0.000, B 0.000, C 0.000 }
gfCNCPoint3[397] = {X 61.5183, Y 7.6903, Z -3.8333, A 0.000, B 0.000, C 0.000 }
gfCNCPoint3[398] = {X 62.3719, Y 8.1553, Z -3.8333, A 0.000, B 0.000, C 0.000 }
gfCNCPoint3[399] = {X 63.1164, Y 8.7803, Z -3.8333, A 0.000, B 0.000, C 0.000 }
gfCNCPoint3[400] = {X 63.7054, Y 9.5145, Z -3.8333, A 0.000, B 0.000, C 0.000 }
gfCNCPoint3[401] = {X 64.1424, Y 10.3480, Z -3.8333, A 0.000, B 0.000, C 0.000 }
gfCNCPoint3[402] = {X 64.4114, Y 11.2500, Z -3.8333, A 0.000, B 0.000, C 0.000 }
gfCNCPoint3[403] = {X 64.5021, Y 12.1868, Z -3.8333, A 0.000, B 0.000, C 0.000 }
gfCNCPoint3[404] = {X 64.5019, Y 13.0237, Z -3.8333, A 0.000, B 0.000, C 0.000 }
gfCNCPoint3[405] = {X 64.4204, Y 13.8675, Z -3.8333, A 0.000, B 0.000, C 0.000 }
gfCNCPoint3[406] = {X 64.1940, Y 14.6844, Z -3.8333, A 0.000, B 0.000, C 0.000 }
gfCNCPoint3[407] = {X 63.8298, Y 15.4499, Z -3.8333, A 0.000, B 0.000, C 0.000 }
gfCNCPoint3[408] = {X 72.9540, Y 39.8577, Z -3.8333, A 0.000, B 0.000, C 0.000 }
gfCNCPoint3[409] = {X 73.8441, Y 40.4396, Z -3.8333, A 0.000, B 0.000, C 0.000 }
gfCNCPoint3[410] = {X 74.5870, Y 41.2005, Z -3.8333, A 0.000, B 0.000, C 0.000 }
gfCNCPoint3[411] = {X 75.1474, Y 42.1043, Z -3.8333, A 0.000, B 0.000, C 0.000 }
gfCNCPoint3[412] = {X 75.4987, Y 43.1080, Z -3.8333, A 0.000, B 0.000, C 0.000 }
gfCNCPoint3[413] = {X 75.6243, Y 44.1640, Z -3.8333, A 0.000, B 0.000, C 0.000 }
gfCNCPoint3[414] = {X 75.6245, Y 45.0000, Z -3.8333, A 0.000, B 0.000, C 0.000 }
gfCNCPoint3[415] = {X 75.5307, Y 45.9520, Z -3.8333, A 0.000, B 0.000, C 0.000 }
gfCNCPoint3[416] = {X 75.2530, Y 46.8675, Z -3.8333, A 0.000, B 0.000, C 0.000 }
gfCNCPoint3[417] = {X 74.8020, Y 47.7112, Z -3.8333, A 0.000, B 0.000, C 0.000 }
gfCNCPoint3[418] = {X 74.1951, Y 48.4507, Z -3.8333, A 0.000, B 0.000, C 0.000 }
gfCNCPoint3[419] = {X 73.4556, Y 49.0576, Z -3.8333, A 0.000, B 0.000, C 0.000 }
gfCNCPoint3[420] = {X 72.6120, Y 49.5085, Z -3.8333, A 0.000, B 0.000, C 0.000 }
gfCNCPoint3[421] = {X 71.6965, Y 49.7862, Z -3.8333, A 0.000, B 0.000, C 0.000 }
gfCNCPoint3[422] = {X 70.7445, Y 49.8800, Z -3.8333, A 0.000, B 0.000, C 0.000 }
gfCNCPoint3[423] = {X 64.1851, Y 49.8800, Z -3.8333, A 0.000, B 0.000, C 0.000 }
gfCNCPoint3[424] = {X 63.2331, Y 49.7862, Z -3.8333, A 0.000, B 0.000, C 0.000 }
gfCNCPoint3[425] = {X 62.3176, Y 49.5085, Z -3.8333, A 0.000, B 0.000, C 0.000 }
gfCNCPoint3[426] = {X 61.4740, Y 49.0576, Z -3.8333, A 0.000, B 0.000, C 0.000 }
gfCNCPoint3[427] = {X 60.7345, Y 48.4507, Z -3.8333, A 0.000, B 0.000, C 0.000 }
gfCNCPoint3[428] = {X 60.1276, Y 47.7112, Z -3.8333, A 0.000, B 0.000, C 0.000 }
gfCNCPoint3[429] = {X 59.6766, Y 46.8675, Z -3.8333, A 0.000, B 0.000, C 0.000 }
gfCNCPoint3[430] = {X 59.3989, Y 45.9520, Z -3.8333, A 0.000, B 0.000, C 0.000 }
gfCNCPoint3[431] = {X 59.3051, Y 45.0000, Z -3.8333, A 0.000, B 0.000, C 0.000 }
gfCNCPoint3[432] = {X 59.3052, Y 44.2029, Z -3.8333, A 0.000, B 0.000, C 0.000 }
gfCNCPoint3[433] = {X 59.3847, Y 43.3310, Z -3.8333, A 0.000, B 0.000, C 0.000 }
gfCNCPoint3[434] = {X 59.6188, Y 42.4874, Z -3.8333, A 0.000, B 0.000, C 0.000 }
gfCNCPoint3[435] = {X 59.9999, Y 41.6992, Z -3.8333, A 0.000, B 0.000, C 0.000 }
gfCNCPoint3[436] = {X 59.6157, Y 40.6492, Z -3.8333, A 0.000, B 0.000, C 0.000 }
gfCNCPoint3[437] = {X 52.4661, Y 40.6492, Z -3.8333, A 0.000, B 0.000, C 0.000 }
gfCNCPoint3[438] = {X 51.9468, Y 42.0445, Z -3.8333, A 0.000, B 0.000, C 0.000 }
gfCNCPoint3[439] = {X 52.2215, Y 42.7239, Z -3.8333, A 0.000, B 0.000, C 0.000 }
gfCNCPoint3[440] = {X 52.3915, Y 43.4369, Z -3.8333, A 0.000, B 0.000, C 0.000 }
gfCNCPoint3[441] = {X 52.4528, Y 44.1672, Z -3.8333, A 0.000, B 0.000, C 0.000 }
gfCNCPoint3[442] = {X 52.4529, Y 45.0000, Z -3.8333, A 0.000, B 0.000, C 0.000 }
gfCNCPoint3[443] = {X 52.3592, Y 45.9520, Z -3.8333, A 0.000, B 0.000, C 0.000 }
gfCNCPoint3[444] = {X 52.0815, Y 46.8675, Z -3.8333, A 0.000, B 0.000, C 0.000 }
gfCNCPoint3[445] = {X 51.6305, Y 47.7112, Z -3.8333, A 0.000, B 0.000, C 0.000 }
gfCNCPoint3[446] = {X 51.0236, Y 48.4507, Z -3.8333, A 0.000, B 0.000, C 0.000 }
gfCNCPoint3[447] = {X 50.2841, Y 49.0576, Z -3.8333, A 0.000, B 0.000, C 0.000 }
gfCNCPoint3[448] = {X 49.4404, Y 49.5085, Z -3.8333, A 0.000, B 0.000, C 0.000 }
gfCNCPoint3[449] = {X 48.5250, Y 49.7862, Z -3.8333, A 0.000, B 0.000, C 0.000 }
gfCNCPoint3[450] = {X 47.5729, Y 49.8800, Z -3.8333, A 0.000, B 0.000, C 0.000 }
gfCNCPoint3[451] = {X 40.6393, Y 49.8800, Z -3.8333, A 0.000, B 0.000, C 0.000 }
gfCNCPoint3[452] = {X 39.6433, Y 49.7773, Z -3.8333, A 0.000, B 0.000, C 0.000 }
gfCNCPoint3[453] = {X 38.6892, Y 49.4734, Z -3.8333, A 0.000, B 0.000, C 0.000 }
gfCNCPoint3[454] = {X 37.8173, Y 48.9813, Z -3.8333, A 0.000, B 0.000, C 0.000 }
gfCNCPoint3[455] = {X 37.0641, Y 48.3215, Z -3.8333, A 0.000, B 0.000, C 0.000 }
gfCNCPoint3[456] = {X 36.5085, Y 47.5983, Z -3.8333, A 0.000, B 0.000, C 0.000 }
gfCNCPoint3[457] = {X 36.0972, Y 46.7843, Z -3.8333, A 0.000, B 0.000, C 0.000 }
gfCNCPoint3[458] = {X 35.8445, Y 45.9080, Z -3.8333, A 0.000, B 0.000, C 0.000 }
gfCNCPoint3[459] = {X 35.7593, Y 45.0000, Z -3.8333, A 0.000, B 0.000, C 0.000 }
gfCNCPoint3[460] = {X 35.7593, Y 44.7148, Z -3.8333, A 0.000, B 0.000, C 0.000 }
gfCNCPoint3[461] = {X 36.2393, Y 44.7148, Z -3.8333, A 0.000, B 0.000, C 0.000 }
gfCNCPoint3[462] = {X 36.2397, Y 44.1483, Z -3.8333, A 0.000, B 0.000, C 0.000 }
gfCNCPoint3[463] = {X 36.3681, Y 43.1521, Z -3.8333, A 0.000, B 0.000, C 0.000 }
gfCNCPoint3[464] = {X 36.7190, Y 42.2110, Z -3.8333, A 0.000, B 0.000, C 0.000 }
gfCNCPoint3[465] = {X 37.2742, Y 41.3740, Z -3.8333, A 0.000, B 0.000, C 0.000 }
gfCNCPoint3[466] = {X 38.0047, Y 40.6847, Z -3.8333, A 0.000, B 0.000, C 0.000 }
gfCNCPoint3[467] = {X 38.8726, Y 40.1791, Z -3.8333, A 0.000, B 0.000, C 0.000 }
gfCNCPoint3[468] = {X 39.4560, Y 38.7987, Z -3.8333, A 0.000, B 0.000, C 0.000 }
gfCNCPoint3[469] = {X 39.9907, Y 37.3987, Z -3.8333, A 0.000, B 0.000, C 0.000 }
gfCNCPoint3[470] = {X 48.2011, Y 15.3544, Z -3.8333, A 0.000, B 0.000, C 0.000 }
gfCNCPoint3[471] = {X 47.8187, Y 14.6115, Z -3.8333, A 0.000, B 0.000, C 0.000 }
gfCNCPoint3[472] = {X 47.5835, Y 13.8097, Z -3.8333, A 0.000, B 0.000, C 0.000 }
gfCNCPoint3[473] = {X 47.5042, Y 12.9779, Z -3.8333, A 0.000, B 0.000, C 0.000 }
gfCNCPoint3[474] = {X 47.5042, Y 12.1868, Z -3.8333, A 0.000, B 0.000, C 0.000 }
gfCNCPoint3[475] = {X 47.6145, Y 11.2077, Z -3.8333, A 0.000, B 0.000, C 0.000 }
gfCNCPoint3[476] = {X 47.9400, Y 10.2777, Z -3.8333, A 0.000, B 0.000, C 0.000 }
gfCNCPoint3[477] = {X 48.4642, Y 9.4435, Z -3.8333, A 0.000, B 0.000, C 0.000 }
gfCNCPoint3[478] = {X 49.1609, Y 8.7468, Z -3.8333, A 0.000, B 0.000, C 0.000 }
gfCNCPoint3[479] = {X 49.9951, Y 8.2226, Z -3.8333, A 0.000, B 0.000, C 0.000 }
gfCNCPoint3[480] = {X 50.9251, Y 7.8971, Z -3.8333, A 0.000, B 0.000, C 0.000 }
gfCNCPoint3[481] = {X 51.9042, Y 7.7868, Z -3.8333, A 0.000, B 0.000, C 0.000 }
gfCNCPoint3[482] = {X 59.6221, Y 7.7868, Z -3.8333, A 0.000, B 0.000, C 0.000 }
gfCNCPoint3[483] = {X 60.6012, Y 7.8971, Z -3.8333, A 0.000, B 0.000, C 0.000 }
gfCNCPoint3[484] = {X 61.5312, Y 8.2226, Z -3.8333, A 0.000, B 0.000, C 0.000 }
gfCNCPoint3[485] = {X 62.3655, Y 8.7468, Z -3.8333, A 0.000, B 0.000, C 0.000 }
gfCNCPoint3[486] = {X 63.0622, Y 9.4435, Z -3.8333, A 0.000, B 0.000, C 0.000 }
gfCNCPoint3[487] = {X 63.5864, Y 10.2777, Z -3.8333, A 0.000, B 0.000, C 0.000 }
gfCNCPoint3[488] = {X 63.9118, Y 11.2077, Z -3.8333, A 0.000, B 0.000, C 0.000 }
gfCNCPoint3[489] = {X 64.0221, Y 12.1868, Z -3.8333, A 0.000, B 0.000, C 0.000 }
gfCNCPoint3[490] = {X 64.0219, Y 13.0233, Z -3.8333, A 0.000, B 0.000, C 0.000 }
gfCNCPoint3[491] = {X 63.9336, Y 13.8564, Z -3.8333, A 0.000, B 0.000, C 0.000 }
gfCNCPoint3[492] = {X 63.6889, Y 14.6577, Z -3.8333, A 0.000, B 0.000, C 0.000 }
gfCNCPoint3[493] = {X 63.2968, Y 15.3981, Z -3.8333, A 0.000, B 0.000, C 0.000 }
gfCNCPoint3[494] = {X 63.5004, Y 15.9354, Z -3.8333, A 0.000, B 0.000, C 0.000 }
gfCNCPoint3[495] = {X 66.3154, Y 23.4043, Z -3.8333, A 0.000, B 0.000, C 0.000 }
gfCNCPoint3[496] = {X 72.2840, Y 39.4717, Z -3.8333, A 0.000, B 0.000, C 0.000 }
gfCNCPoint3[497] = {X 72.5770, Y 40.2086, Z -3.8333, A 0.000, B 0.000, C 0.000 }
gfCNCPoint3[498] = {X 73.4346, Y 40.7270, Z -3.8333, A 0.000, B 0.000, C 0.000 }
gfCNCPoint3[499] = {X 74.1527, Y 41.4260, Z -3.8333, A 0.000, B 0.000, C 0.000 }
gfCNCPoint3[500] = {X 74.6940, Y 42.2693, Z -3.8333, A 0.000, B 0.000, C 0.000 }
gfCNCPoint3[501] = {X 75.0304, Y 43.2133, Z -3.8333, A 0.000, B 0.000, C 0.000 }
gfCNCPoint3[502] = {X 75.1445, Y 44.2089, Z -3.8333, A 0.000, B 0.000, C 0.000 }
gfCNCPoint3[503] = {X 75.1445, Y 45.0000, Z -3.8333, A 0.000, B 0.000, C 0.000 }
gfCNCPoint3[504] = {X 75.0341, Y 45.9791, Z -3.8333, A 0.000, B 0.000, C 0.000 }
gfCNCPoint3[505] = {X 74.7087, Y 46.9091, Z -3.8333, A 0.000, B 0.000, C 0.000 }
gfCNCPoint3[506] = {X 74.1845, Y 47.7434, Z -3.8333, A 0.000, B 0.000, C 0.000 }
gfCNCPoint3[507] = {X 73.4878, Y 48.4401, Z -3.8333, A 0.000, B 0.000, C 0.000 }
gfCNCPoint3[508] = {X 72.6535, Y 48.9643, Z -3.8333, A 0.000, B 0.000, C 0.000 }
gfCNCPoint3[509] = {X 71.7236, Y 49.2897, Z -3.8333, A 0.000, B 0.000, C 0.000 }
gfCNCPoint3[510] = {X 70.7445, Y 49.4000, Z -3.8333, A 0.000, B 0.000, C 0.000 }
gfCNCPoint3[511] = {X 64.1851, Y 49.4000, Z -3.8333, A 0.000, B 0.000, C 0.000 }
gfCNCPoint3[512] = {X 63.2060, Y 49.2897, Z -3.8333, A 0.000, B 0.000, C 0.000 }
gfCNCPoint3[513] = {X 62.2760, Y 48.9643, Z -3.8333, A 0.000, B 0.000, C 0.000 }
gfCNCPoint3[514] = {X 61.4418, Y 48.4401, Z -3.8333, A 0.000, B 0.000, C 0.000 }
gfCNCPoint3[515] = {X 60.7451, Y 47.7434, Z -3.8333, A 0.000, B 0.000, C 0.000 }
gfCNCPoint3[516] = {X 60.2209, Y 46.9091, Z -3.8333, A 0.000, B 0.000, C 0.000 }
gfCNCPoint3[517] = {X 59.8955, Y 45.9791, Z -3.8333, A 0.000, B 0.000, C 0.000 }
gfCNCPoint3[518] = {X 59.7851, Y 45.0000, Z -3.8333, A 0.000, B 0.000, C 0.000 }
gfCNCPoint3[519] = {X 59.7856, Y 44.1483, Z -3.8333, A 0.000, B 0.000, C 0.000 }
gfCNCPoint3[520] = {X 59.8784, Y 43.3077, Z -3.8333, A 0.000, B 0.000, C 0.000 }
gfCNCPoint3[521] = {X 60.1303, Y 42.5005, Z -3.8333, A 0.000, B 0.000, C 0.000 }
gfCNCPoint3[522] = {X 60.5320, Y 41.7564, Z -3.8333, A 0.000, B 0.000, C 0.000 }
gfCNCPoint3[523] = {X 59.9512, Y 40.1692, Z -3.8333, A 0.000, B 0.000, C 0.000 }
gfCNCPoint3[524] = {X 52.1326, Y 40.1692, Z -3.8333, A 0.000, B 0.000, C 0.000 }
gfCNCPoint3[525] = {X 51.4223, Y 42.0775, Z -3.8333, A 0.000, B 0.000, C 0.000 }
gfCNCPoint3[526] = {X 51.7253, Y 42.7535, Z -3.8333, A 0.000, B 0.000, C 0.000 }
gfCNCPoint3[527] = {X 51.9106, Y 43.4707, Z -3.8333, A 0.000, B 0.000, C 0.000 }
gfCNCPoint3[528] = {X 51.9729, Y 44.2089, Z -3.8333, A 0.000, B 0.000, C 0.000 }
gfCNCPoint3[529] = {X 51.9729, Y 45.0000, Z -3.8333, A 0.000, B 0.000, C 0.000 }
gfCNCPoint3[530] = {X 51.8626, Y 45.9791, Z -3.8333, A 0.000, B 0.000, C 0.000 }
gfCNCPoint3[531] = {X 51.5372, Y 46.9091, Z -3.8333, A 0.000, B 0.000, C 0.000 }
gfCNCPoint3[532] = {X 51.0130, Y 47.7434, Z -3.8333, A 0.000, B 0.000, C 0.000 }
gfCNCPoint3[533] = {X 50.3163, Y 48.4401, Z -3.8333, A 0.000, B 0.000, C 0.000 }
gfCNCPoint3[534] = {X 49.4820, Y 48.9643, Z -3.8333, A 0.000, B 0.000, C 0.000 }
gfCNCPoint3[535] = {X 48.5520, Y 49.2897, Z -3.8333, A 0.000, B 0.000, C 0.000 }
gfCNCPoint3[536] = {X 47.5729, Y 49.4000, Z -3.8333, A 0.000, B 0.000, C 0.000 }
gfCNCPoint3[537] = {X 40.6393, Y 49.4000, Z -3.8333, A 0.000, B 0.000, C 0.000 }
gfCNCPoint3[538] = {X 39.6602, Y 49.2897, Z -3.8333, A 0.000, B 0.000, C 0.000 }
gfCNCPoint3[539] = {X 38.7302, Y 48.9643, Z -3.8333, A 0.000, B 0.000, C 0.000 }
gfCNCPoint3[540] = {X 37.8959, Y 48.4401, Z -3.8333, A 0.000, B 0.000, C 0.000 }
gfCNCPoint3[541] = {X 37.1992, Y 47.7434, Z -3.8333, A 0.000, B 0.000, C 0.000 }
gfCNCPoint3[542] = {X 36.6750, Y 46.9091, Z -3.8333, A 0.000, B 0.000, C 0.000 }
gfCNCPoint3[543] = {X 36.3496, Y 45.9791, Z -3.8333, A 0.000, B 0.000, C 0.000 }
gfCNCPoint3[544] = {X 36.2393, Y 45.0000, Z -3.8333, A 0.000, B 0.000, C 0.000 }
gfCNCPoint3[545] = {X 36.2393, Y 44.7148, Z -3.8333, A 0.000, B 0.000, C 0.000 }
gfCNCPoint3[546] = {X 35.7593, Y 44.7148, Z -3.8333, A 0.000, B 0.000, C 0.000 }
gfCNCPoint3[547] = {X 35.2211, Y 46.0074, Z -3.8333, A 0.000, B 0.000, C 0.000 }
gfCNCPoint3[548] = {X 34.4930, Y 47.2034, Z -3.8333, A 0.000, B 0.000, C 0.000 }
gfCNCPoint3[549] = {X 33.5918, Y 48.2750, Z -3.8333, A 0.000, B 0.000, C 0.000 }
gfCNCPoint3[550] = {X 33.2092, Y 48.6435, Z -3.8333, A 0.000, B 0.000, C 0.000 }
gfCNCPoint3[551] = {X 32.8060, Y 48.9892, Z -3.8333, A 0.000, B 0.000, C 0.000 }
gfCNCPoint3[552] = {X 32.2668, Y 49.4252, Z -3.8333, A 0.000, B 0.000, C 0.000 }
gfCNCPoint3[553] = {X 31.1805, Y 50.1801, Z -3.8333, A 0.000, B 0.000, C 0.000 }
gfCNCPoint3[554] = {X 29.9974, Y 50.7716, Z -3.8333, A 0.000, B 0.000, C 0.000 }
gfCNCPoint3[555] = {X 28.7417, Y 51.1877, Z -3.8333, A 0.000, B 0.000, C 0.000 }
gfCNCPoint3[556] = {X 27.4394, Y 51.4198, Z -3.8333, A 0.000, B 0.000, C 0.000 }
gfCNCPoint3[557] = {X 26.1173, Y 51.4629, Z -3.8333, A 0.000, B 0.000, C 0.000 }
gfCNCPoint3[558] = {X 23.6803, Y 52.5818, Z -3.8333, A 0.000, B 0.000, C 0.000 }
gfCNCPoint3[559] = {X 21.1625, Y 53.5046, Z -3.8333, A 0.000, B 0.000, C 0.000 }
gfCNCPoint3[560] = {X 18.9475, Y 54.1336, Z -3.8333, A 0.000, B 0.000, C 0.000 }
gfCNCPoint3[561] = {X 16.6881, Y 54.5767, Z -3.8333, A 0.000, B 0.000, C 0.000 }
gfCNCPoint3[562] = {X 14.3996, Y 54.8309, Z -3.8333, A 0.000, B 0.000, C 0.000 }
gfCNCPoint3[563] = {X 12.0980, Y 54.8943, Z -3.8333, A 0.000, B 0.000, C 0.000 }
gfCNCPoint3[564] = {X 9.7991, Y 54.7666, Z -3.8333, A 0.000, B 0.000, C 0.000 }
gfCNCPoint3[565] = {X 7.5186, Y 54.4486, Z -3.8333, A 0.000, B 0.000, C 0.000 }
gfCNCPoint3[566] = {X 6.0997, Y 54.1508, Z -3.8333, A 0.000, B 0.000, C 0.000 }
gfCNCPoint3[567] = {X 4.7035, Y 53.7601, Z -3.8333, A 0.000, B 0.000, C 0.000 }
gfCNCPoint3[568] = {X 4.7035, Y 95.2950, Z -3.8333, A 0.000, B 0.000, C 0.000 }
gfCNCPoint3[569] = {X 117.9387, Y 95.2950, Z -3.8333, A 0.000, B 0.000, C 0.000 }
gfCNCPoint3[570] = {X 118.3614, Y 94.0781, Z -3.8333, A 0.000, B 0.000, C 0.000 }
gfCNCPoint3[571] = {X 118.9919, Y 92.9548, Z -3.8333, A 0.000, B 0.000, C 0.000 }
gfCNCPoint3[572] = {X 119.8106, Y 91.9602, Z -3.8333, A 0.000, B 0.000, C 0.000 }
gfCNCPoint3[573] = {X 120.7918, Y 91.1255, Z -3.8333, A 0.000, B 0.000, C 0.000 }
gfCNCPoint3[574] = {X 121.9047, Y 90.4767, Z -3.8333, A 0.000, B 0.000, C 0.000 }
gfCNCPoint3[575] = {X 123.1146, Y 90.0343, Z -3.8333, A 0.000, B 0.000, C 0.000 }
gfCNCPoint3[576] = {X 124.3835, Y 89.8121, Z -3.8333, A 0.000, B 0.000, C 0.000 }
gfCNCPoint3[577] = {X 124.4935, Y 89.7938, Z -3.8333, A 0.000, B 0.000, C 0.000 }
gfCNCPoint3[578] = {X 125.0314, Y 89.7140, Z -3.8333, A 0.000, B 0.000, C 0.000 }
gfCNCPoint3[579] = {X 125.3489, Y 89.6671, Z -3.8333, A 0.000, B 0.000, C 0.000 }
gfCNCPoint3[580] = {X 125.6646, Y 89.6093, Z -3.8333, A 0.000, B 0.000, C 0.000 }
gfCNCPoint3[581] = {X 126.4917, Y 88.7985, Z -3.8333, A 0.000, B 0.000, C 0.000 }
gfCNCPoint3[582] = {X 127.2845, Y 87.9541, Z -3.8333, A 0.000, B 0.000, C 0.000 }
gfCNCPoint3[583] = {X 152.2076, Y 60.5850, Z -3.8333, A 0.000, B 0.000, C 0.000 }
gfCNCPoint3[584] = {X 152.0684, Y 59.7900, Z -3.8333, A 0.000, B 0.000, C 0.000 }
gfCNCPoint3[585] = {X 152.0181, Y 58.9845, Z -3.8333, A 0.000, B 0.000, C 0.000 }
gfCNCPoint3[586] = {X 152.0180, Y 58.0000, Z -3.8333, A 0.000, B 0.000, C 0.000 }
gfCNCPoint3[587] = {X 152.1286, Y 56.7358, Z -3.8333, A 0.000, B 0.000, C 0.000 }
gfCNCPoint3[588] = {X 152.4570, Y 55.5101, Z -3.8333, A 0.000, B 0.000, C 0.000 }
gfCNCPoint3[589] = {X 152.9933, Y 54.3600, Z -3.8333, A 0.000, B 0.000, C 0.000 }
gfCNCPoint3[590] = {X 153.7212, Y 53.3205, Z -3.8333, A 0.000, B 0.000, C 0.000 }
gfCNCPoint3[591] = {X 154.6185, Y 52.4232, Z -3.8333, A 0.000, B 0.000, C 0.000 }
gfCNCPoint3[592] = {X 155.6580, Y 51.6953, Z -3.8333, A 0.000, B 0.000, C 0.000 }
gfCNCPoint3[593] = {X 156.8081, Y 51.1590, Z -3.8333, A 0.000, B 0.000, C 0.000 }
gfCNCPoint3[594] = {X 158.0338, Y 50.8306, Z -3.8333, A 0.000, B 0.000, C 0.000 }
gfCNCPoint3[595] = {X 159.2980, Y 50.7200, Z -3.8333, A 0.000, B 0.000, C 0.000 }
gfCNCPoint3[596] = {X 178.5335, Y 50.7200, Z -3.8333, A 0.000, B 0.000, C 0.000 }
gfCNCPoint3[597] = {X 179.7869, Y 50.8287, Z -3.8333, A 0.000, B 0.000, C 0.000 }
gfCNCPoint3[598] = {X 181.0029, Y 51.1516, Z -3.8333, A 0.000, B 0.000, C 0.000 }
gfCNCPoint3[599] = {X 182.1451, Y 51.6790, Z -3.8333, A 0.000, B 0.000, C 0.000 }
gfCNCPoint3[600] = {X 183.1795, Y 52.3953, Z -3.8333, A 0.000, B 0.000, C 0.000 }
gfCNCPoint3[601] = {X 184.0878, Y 53.2938, Z -3.8333, A 0.000, B 0.000, C 0.000 }
gfCNCPoint3[602] = {X 184.8250, Y 54.3374, Z -3.8333, A 0.000, B 0.000, C 0.000 }
gfCNCPoint3[603] = {X 185.3685, Y 55.4937, Z -3.8333, A 0.000, B 0.000, C 0.000 }
gfCNCPoint3[604] = {X 185.7014, Y 56.7273, Z -3.8333, A 0.000, B 0.000, C 0.000 }
gfCNCPoint3[605] = {X 185.8135, Y 58.0000, Z -3.8333, A 0.000, B 0.000, C 0.000 }
gfCNCPoint3[606] = {X 185.8133, Y 58.9942, Z -3.8333, A 0.000, B 0.000, C 0.000 }
gfCNCPoint3[607] = {X 185.7648, Y 59.7751, Z -3.8333, A 0.000, B 0.000, C 0.000 }
gfCNCPoint3[608] = {X 185.6327, Y 60.5463, Z -3.8333, A 0.000, B 0.000, C 0.000 }
gfCNCPoint3[609] = {X 211.6608, Y 88.9544, Z -3.8333, A 0.000, B 0.000, C 0.000 }
gfCNCPoint3[610] = {X 212.0331, Y 89.3393, Z -3.8333, A 0.000, B 0.000, C 0.000 }
gfCNCPoint3[611] = {X 212.4256, Y 89.7034, Z -3.8333, A 0.000, B 0.000, C 0.000 }
gfCNCPoint3[612] = {X 212.6034, Y 89.7414, Z -3.8333, A 0.000, B 0.000, C 0.000 }
gfCNCPoint3[613] = {X 213.4472, Y 89.8477, Z -3.8333, A 0.000, B 0.000, C 0.000 }
gfCNCPoint3[614] = {X 214.4297, Y 89.7709, Z -3.8333, A 0.000, B 0.000, C 0.000 }
gfCNCPoint3[615] = {X 215.4136, Y 89.7172, Z -3.8333, A 0.000, B 0.000, C 0.000 }
gfCNCPoint3[616] = {X 215.6262, Y 89.6937, Z -3.8333, A 0.000, B 0.000, C 0.000 }
gfCNCPoint3[617] = {X 215.8216, Y 89.6067, Z -3.8333, A 0.000, B 0.000, C 0.000 }
gfCNCPoint3[618] = {X 239.3466, Y 74.5356, Z -3.8333, A 0.000, B 0.000, C 0.000 }
gfCNCPoint3[619] = {X 220.5435, Y 67.1566, Z -3.8333, A 0.000, B 0.000, C 0.000 }
gfCNCPoint3[620] = {X 219.0952, Y 66.6703, Z -3.8333, A 0.000, B 0.000, C 0.000 }
gfCNCPoint3[621] = {X 217.6006, Y 66.3533, Z -3.8333, A 0.000, B 0.000, C 0.000 }
gfCNCPoint3[622] = {X 216.0796, Y 66.2097, Z -3.8333, A 0.000, B 0.000, C 0.000 }
gfCNCPoint3[623] = {X 214.8528, Y 66.0624, Z -3.8333, A 0.000, B 0.000, C 0.000 }
gfCNCPoint3[624] = {X 213.6686, Y 65.7098, Z -3.8333, A 0.000, B 0.000, C 0.000 }
gfCNCPoint3[625] = {X 212.5611, Y 65.1620, Z -3.8333, A 0.000, B 0.000, C 0.000 }
gfCNCPoint3[626] = {X 211.5621, Y 64.4348, Z -3.8333, A 0.000, B 0.000, C 0.000 }
gfCNCPoint3[627] = {X 210.7006, Y 63.5492, Z -3.8333, A 0.000, B 0.000, C 0.000 }
gfCNCPoint3[628] = {X 210.0012, Y 62.5305, Z -3.8333, A 0.000, B 0.000, C 0.000 }
gfCNCPoint3[629] = {X 209.4842, Y 61.4083, Z -3.8333, A 0.000, B 0.000, C 0.000 }
gfCNCPoint3[630] = {X 209.1644, Y 60.2149, Z -3.8333, A 0.000, B 0.000, C 0.000 }
gfCNCPoint3[631] = {X 209.0510, Y 58.9845, Z -3.8333, A 0.000, B 0.000, C 0.000 }
gfCNCPoint3[632] = {X 209.0508, Y 58.0000, Z -3.8333, A 0.000, B 0.000, C 0.000 }
gfCNCPoint3[633] = {X 209.1477, Y 56.8162, Z -3.8333, A 0.000, B 0.000, C 0.000 }
gfCNCPoint3[634] = {X 209.4358, Y 55.6638, Z -3.8333, A 0.000, B 0.000, C 0.000 }
gfCNCPoint3[635] = {X 209.9075, Y 54.5737, Z -3.8333, A 0.000, B 0.000, C 0.000 }
gfCNCPoint3[636] = {X 210.5502, Y 53.5748, Z -3.8333, A 0.000, B 0.000, C 0.000 }
gfCNCPoint3[637] = {X 211.3467, Y 52.6937, Z -3.8333, A 0.000, B 0.000, C 0.000 }
gfCNCPoint3[638] = {X 212.2759, Y 51.9538, Z -3.8333, A 0.000, B 0.000, C 0.000 }
gfCNCPoint3[639] = {X 213.3131, Y 51.3749, Z -3.8333, A 0.000, B 0.000, C 0.000 }
gfCNCPoint3[640] = {X 214.4306, Y 50.9724, Z -3.8333, A 0.000, B 0.000, C 0.000 }
gfCNCPoint3[641] = {X 215.3724, Y 50.7834, Z -3.8333, A 0.000, B 0.000, C 0.000 }
gfCNCPoint3[642] = {X 216.3308, Y 50.7200, Z -3.8333, A 0.000, B 0.000, C 0.000 }
gfCNCPoint3[643] = {X 237.2617, Y 50.7200, Z -3.8333, A 0.000, B 0.000, C 0.000 }
gfCNCPoint3[644] = {X 238.3057, Y 50.7953, Z -3.8333, A 0.000, B 0.000, C 0.000 }
gfCNCPoint3[645] = {X 239.3282, Y 51.0195, Z -3.8333, A 0.000, B 0.000, C 0.000 }
gfCNCPoint3[646] = {X 240.3080, Y 51.3880, Z -3.8333, A 0.000, B 0.000, C 0.000 }
gfCNCPoint3[647] = {X 241.2247, Y 51.8932, Z -3.8333, A 0.000, B 0.000, C 0.000 }
gfCNCPoint3[648] = {X 242.0741, Y 52.5375, Z -3.8333, A 0.000, B 0.000, C 0.000 }
gfCNCPoint3[649] = {X 242.8203, Y 53.2989, Z -3.8333, A 0.000, B 0.000, C 0.000 }
gfCNCPoint3[650] = {X 243.4473, Y 54.1611, Z -3.8333, A 0.000, B 0.000, C 0.000 }
gfCNCPoint3[651] = {X 243.9416, Y 55.1057, Z -3.8333, A 0.000, B 0.000, C 0.000 }
gfCNCPoint3[652] = {X 244.2927, Y 56.1123, Z -3.8333, A 0.000, B 0.000, C 0.000 }
gfCNCPoint3[653] = {X 248.5777, Y 57.7827, Z -3.8333, A 0.000, B 0.000, C 0.000 }
gfCNCPoint3[654] = {X 272.6728, Y 67.3433, Z -3.8333, A 0.000, B 0.000, C 0.000 }
gfCNCPoint3[655] = {X 272.6727, Y 65.2842, Z -3.8333, A 0.000, B 0.000, C 0.000 }
gfCNCPoint3[656] = {X 271.6654, Y 64.6031, Z -3.8333, A 0.000, B 0.000, C 0.000 }
gfCNCPoint3[657] = {X 270.7855, Y 63.7638, Z -3.8333, A 0.000, B 0.000, C 0.000 }
gfCNCPoint3[658] = {X 270.0576, Y 62.7898, Z -3.8333, A 0.000, B 0.000, C 0.000 }
gfCNCPoint3[659] = {X 269.5019, Y 61.7082, Z -3.8333, A 0.000, B 0.000, C 0.000 }
gfCNCPoint3[660] = {X 269.2029, Y 60.8262, Z -3.8333, A 0.000, B 0.000, C 0.000 }
gfCNCPoint3[661] = {X 269.0189, Y 59.9134, Z -3.8333, A 0.000, B 0.000, C 0.000 }
gfCNCPoint3[662] = {X 268.9529, Y 58.9845, Z -3.8333, A 0.000, B 0.000, C 0.000 }
gfCNCPoint3[663] = {X 268.9527, Y 58.0000, Z -3.8333, A 0.000, B 0.000, C 0.000 }
gfCNCPoint3[664] = {X 269.0633, Y 56.7358, Z -3.8333, A 0.000, B 0.000, C 0.000 }
gfCNCPoint3[665] = {X 269.3917, Y 55.5101, Z -3.8333, A 0.000, B 0.000, C 0.000 }
gfCNCPoint3[666] = {X 269.9280, Y 54.3600, Z -3.8333, A 0.000, B 0.000, C 0.000 }
gfCNCPoint3[667] = {X 270.6559, Y 53.3205, Z -3.8333, A 0.000, B 0.000, C 0.000 }
gfCNCPoint3[668] = {X 271.5532, Y 52.4232, Z -3.8333, A 0.000, B 0.000, C 0.000 }
gfCNCPoint3[669] = {X 272.5927, Y 51.6953, Z -3.8333, A 0.000, B 0.000, C 0.000 }
gfCNCPoint3[670] = {X 273.7428, Y 51.1590, Z -3.8333, A 0.000, B 0.000, C 0.000 }
gfCNCPoint3[671] = {X 274.9685, Y 50.8306, Z -3.8333, A 0.000, B 0.000, C 0.000 }
gfCNCPoint3[672] = {X 276.2327, Y 50.7200, Z -3.8333, A 0.000, B 0.000, C 0.000 }
gfCNCPoint3[673] = {X 292.7731, Y 50.7200, Z -3.8333, A 0.000, B 0.000, C 0.000 }
gfCNCPoint3[674] = {X 293.4209, Y 50.7489, Z -3.8333, A 0.000, B 0.000, C 0.000 }
gfCNCPoint3[675] = {X 294.0636, Y 50.8353, Z -3.8333, A 0.000, B 0.000, C 0.000 }
gfCNCPoint3[676] = {X 294.7295, Y 50.9878, Z -3.8333, A 0.000, B 0.000, C 0.000 }
gfCNCPoint3[677] = {X 295.3781, Y 51.2020, Z -3.8333, A 0.000, B 0.000, C 0.000 }
gfCNCPoint3[678] = {X 298.3089, Y 43.5541, Z -3.8333, A 0.000, B 0.000, C 0.000 }
gfCNCPoint3[679] = {X 298.4822, Y 42.5305, Z -3.8333, A 0.000, B 0.000, C 0.000 }
gfCNCPoint3[680] = {X 298.7927, Y 41.5399, Z -3.8333, A 0.000, B 0.000, C 0.000 }
gfCNCPoint3[681] = {X 299.2347, Y 40.6005, Z -3.8333, A 0.000, B 0.000, C 0.000 }
gfCNCPoint3[682] = {X 299.8001, Y 39.7298, Z -3.8333, A 0.000, B 0.000, C 0.000 }
gfCNCPoint3[683] = {X 299.8001, Y 36.9943, Z -3.8333, A 0.000, B 0.000, C 0.000 }
gfCNCPoint3[684] = {X 296.8139, Y 36.9943, Z -3.8333, A 0.000, B 0.000, C 0.000 }
gfCNCPoint3[685] = {X 296.8135, Y 39.7487, Z -3.8333, A 0.000, B 0.000, C 0.000 }
gfCNCPoint3[686] = {X 297.3849, Y 40.6115, Z -3.8333, A 0.000, B 0.000, C 0.000 }
gfCNCPoint3[687] = {X 297.8300, Y 41.5458, Z -3.8333, A 0.000, B 0.000, C 0.000 }
gfCNCPoint3[688] = {X 298.1400, Y 42.5331, Z -3.8333, A 0.000, B 0.000, C 0.000 }
gfCNCPoint3[689] = {X 298.3089, Y 43.5541, Z -3.8333, A 0.000, B 0.000, C 0.000 }
gfCNCPoint3[690] = {X 296.2369, Y 48.9610, Z -3.8333, A 0.000, B 0.000, C 0.000 }
gfCNCPoint3[691] = {X 296.6127, Y 49.1141, Z -3.8333, A 0.000, B 0.000, C 0.000 }
gfCNCPoint3[692] = {X 296.9817, Y 49.2828, Z -3.8333, A 0.000, B 0.000, C 0.000 }
gfCNCPoint3[693] = {X 297.2571, Y 49.4212, Z -3.8333, A 0.000, B 0.000, C 0.000 }
gfCNCPoint3[694] = {X 297.5280, Y 49.5683, Z -3.8333, A 0.000, B 0.000, C 0.000 }
gfCNCPoint3[695] = {X 298.7174, Y 50.3602, Z -3.8333, A 0.000, B 0.000, C 0.000 }
gfCNCPoint3[696] = {X 299.7774, Y 51.3185, Z -3.8333, A 0.000, B 0.000, C 0.000 }
gfCNCPoint3[697] = {X 300.6847, Y 52.4224, Z -3.8333, A 0.000, B 0.000, C 0.000 }
gfCNCPoint3[698] = {X 301.5914, Y 51.3191, Z -3.8333, A 0.000, B 0.000, C 0.000 }
gfCNCPoint3[699] = {X 302.6506, Y 50.3611, Z -3.8333, A 0.000, B 0.000, C 0.000 }
gfCNCPoint3[700] = {X 303.8393, Y 49.5695, Z -3.8333, A 0.000, B 0.000, C 0.000 }
gfCNCPoint3[701] = {X 302.8989, Y 49.0956, Z -3.8333, A 0.000, B 0.000, C 0.000 }
gfCNCPoint3[702] = {X 302.0820, Y 48.4310, Z -3.8333, A 0.000, B 0.000, C 0.000 }
gfCNCPoint3[703] = {X 301.4268, Y 47.6067, Z -3.8333, A 0.000, B 0.000, C 0.000 }
gfCNCPoint3[704] = {X 300.9636, Y 46.6610, Z -3.8333, A 0.000, B 0.000, C 0.000 }
gfCNCPoint3[705] = {X 300.7923, Y 46.0759, Z -3.8333, A 0.000, B 0.000, C 0.000 }
gfCNCPoint3[706] = {X 300.6953, Y 45.4741, Z -3.8333, A 0.000, B 0.000, C 0.000 }
gfCNCPoint3[707] = {X 300.6790, Y 45.2570, Z -3.8333, A 0.000, B 0.000, C 0.000 }
gfCNCPoint3[708] = {X 300.6724, Y 45.0393, Z -3.8333, A 0.000, B 0.000, C 0.000 }
gfCNCPoint3[709] = {X 300.6725, Y 44.1877, Z -3.8333, A 0.000, B 0.000, C 0.000 }
gfCNCPoint3[710] = {X 300.6810, Y 43.9901, Z -3.8333, A 0.000, B 0.000, C 0.000 }
gfCNCPoint3[711] = {X 300.6970, Y 43.7929, Z -3.8333, A 0.000, B 0.000, C 0.000 }
gfCNCPoint3[712] = {X 300.8618, Y 42.9133, Z -3.8333, A 0.000, B 0.000, C 0.000 }
gfCNCPoint3[713] = {X 301.1740, Y 42.0746, Z -3.8333, A 0.000, B 0.000, C 0.000 }
gfCNCPoint3[714] = {X 301.6245, Y 41.3013, Z -3.8333, A 0.000, B 0.000, C 0.000 }
gfCNCPoint3[715] = {X 302.2001, Y 40.6160, Z -3.8333, A 0.000, B 0.000, C 0.000 }
gfCNCPoint3[716] = {X 302.2001, Y 34.5943, Z -3.8333, A 0.000, B 0.000, C 0.000 }
gfCNCPoint3[717] = {X 294.4142, Y 34.5943, Z -3.8333, A 0.000, B 0.000, C 0.000 }
gfCNCPoint3[718] = {X 294.4134, Y 40.6556, Z -3.8333, A 0.000, B 0.000, C 0.000 }
gfCNCPoint3[719] = {X 294.9938, Y 41.3227, Z -3.8333, A 0.000, B 0.000, C 0.000 }
gfCNCPoint3[720] = {X 295.4470, Y 42.0818, Z -3.8333, A 0.000, B 0.000, C 0.000 }
gfCNCPoint3[721] = {X 295.7588, Y 42.9092, Z -3.8333, A 0.000, B 0.000, C 0.000 }
gfCNCPoint3[722] = {X 295.9194, Y 43.7787, Z -3.8333, A 0.000, B 0.000, C 0.000 }
gfCNCPoint3[723] = {X 295.9349, Y 43.9936, Z -3.8333, A 0.000, B 0.000, C 0.000 }
gfCNCPoint3[724] = {X 295.9411, Y 44.2089, Z -3.8333, A 0.000, B 0.000, C 0.000 }
gfCNCPoint3[725] = {X 295.9411, Y 45.0000, Z -3.8333, A 0.000, B 0.000, C 0.000 }
gfCNCPoint3[726] = {X 295.9354, Y 45.2373, Z -3.8333, A 0.000, B 0.000, C 0.000 }
gfCNCPoint3[727] = {X 295.9181, Y 45.4741, Z -3.8333, A 0.000, B 0.000, C 0.000 }
gfCNCPoint3[728] = {X 298.3067, Y 45.7073, Z -3.8333, A 0.000, B 0.000, C 0.000 }
gfCNCPoint3[729] = {X 298.2010, Y 46.4214, Z -3.8333, A 0.000, B 0.000, C 0.000 }
gfCNCPoint3[730] = {X 298.0252, Y 47.1215, Z -3.8333, A 0.000, B 0.000, C 0.000 }
gfCNCPoint3[731] = {X 298.3689, Y 47.2942, Z -3.8333, A 0.000, B 0.000, C 0.000 }
gfCNCPoint3[732] = {X 298.7069, Y 47.4778, Z -3.8333, A 0.000, B 0.000, C 0.000 }
gfCNCPoint3[733] = {X 298.4514, Y 46.6051, Z -3.8333, A 0.000, B 0.000, C 0.000 }
gfCNCPoint3[734] = {X 298.3067, Y 45.7073, Z -3.8333, A 0.000, B 0.000, C 0.000 }
gfCNCPoint3[735] = {X 295.9181, Y 45.4741, Z -3.8333, A 0.000, B 0.000, C 0.000 }
gfCNCPoint3[736] = {X 295.8472, Y 45.9528, Z -3.8333, A 0.000, B 0.000, C 0.000 }
gfCNCPoint3[737] = {X 295.7293, Y 46.4221, Z -3.8333, A 0.000, B 0.000, C 0.000 }
gfCNCPoint3[738] = {X 295.4314, Y 47.1714, Z -3.8333, A 0.000, B 0.000, C 0.000 }
gfCNCPoint3[739] = {X 295.0142, Y 47.8614, Z -3.8333, A 0.000, B 0.000, C 0.000 }
gfCNCPoint3[740] = {X 294.4890, Y 48.4733, Z -3.8333, A 0.000, B 0.000, C 0.000 }
gfCNCPoint3[741] = {X 295.3744, Y 48.6761, Z -3.8333, A 0.000, B 0.000, C 0.000 }
gfCNCPoint3[742] = {X 296.2369, Y 48.9610, Z -3.8333, A 0.000, B 0.000, C 0.000 }
gfCNCPoint3[743] = {X 295.3781, Y 51.2020, Z -3.8333, A 0.000, B 0.000, C 0.000 }
gfCNCPoint3[744] = {X 296.3501, Y 51.6594, Z -3.8333, A 0.000, B 0.000, C 0.000 }
gfCNCPoint3[745] = {X 297.2443, Y 52.2548, Z -3.8333, A 0.000, B 0.000, C 0.000 }
gfCNCPoint3[746] = {X 298.0410, Y 52.9754, Z -3.8333, A 0.000, B 0.000, C 0.000 }
gfCNCPoint3[747] = {X 298.7231, Y 53.8053, Z -3.8333, A 0.000, B 0.000, C 0.000 }
gfCNCPoint3[748] = {X 299.2946, Y 54.7645, Z -3.8333, A 0.000, B 0.000, C 0.000 }
gfCNCPoint3[749] = {X 299.7126, Y 55.7997, Z -3.8333, A 0.000, B 0.000, C 0.000 }
gfCNCPoint3[750] = {X 299.9675, Y 56.8868, Z -3.8333, A 0.000, B 0.000, C 0.000 }
gfCNCPoint3[751] = {X 300.0531, Y 58.0000, Z -3.8333, A 0.000, B 0.000, C 0.000 }
gfCNCPoint3[752] = {X 300.0531, Y 58.9448, Z -3.8333, A 0.000, B 0.000, C 0.000 }
gfCNCPoint3[753] = {X 299.9646, Y 60.0543, Z -3.8333, A 0.000, B 0.000, C 0.000 }
gfCNCPoint3[754] = {X 299.7084, Y 61.1375, Z -3.8333, A 0.000, B 0.000, C 0.000 }
gfCNCPoint3[755] = {X 299.2904, Y 62.1691, Z -3.8333, A 0.000, B 0.000, C 0.000 }
gfCNCPoint3[756] = {X 298.7203, Y 63.1251, Z -3.8333, A 0.000, B 0.000, C 0.000 }
gfCNCPoint3[757] = {X 300.6820, Y 64.5078, Z -3.8333, A 0.000, B 0.000, C 0.000 }
gfCNCPoint3[758] = {X 299.7823, Y 65.6041, Z -3.8333, A 0.000, B 0.000, C 0.000 }
gfCNCPoint3[759] = {X 298.7324, Y 66.5574, Z -3.8333, A 0.000, B 0.000, C 0.000 }
gfCNCPoint3[760] = {X 298.7324, Y 89.4422, Z -3.8333, A 0.000, B 0.000, C 0.000 }
gfCNCPoint3[761] = {X 299.8291, Y 90.4465, Z -3.8333, A 0.000, B 0.000, C 0.000 }
gfCNCPoint3[762] = {X 300.7597, Y 91.6065, Z -3.8333, A 0.000, B 0.000, C 0.000 }
gfCNCPoint3[763] = {X 301.5022, Y 92.8950, Z -3.8333, A 0.000, B 0.000, C 0.000 }
gfCNCPoint3[764] = {X 304.0674, Y 92.8950, Z -3.8333, A 0.000, B 0.000, C 0.000 }
gfCNCPoint3[765] = {X 303.7098, Y 91.8998, Z -3.8333, A 0.000, B 0.000, C 0.000 }
gfCNCPoint3[766] = {X 303.4138, Y 90.8846, Z -3.8333, A 0.000, B 0.000, C 0.000 }
gfCNCPoint3[767] = {X 302.9747, Y 88.8141, Z -3.8333, A 0.000, B 0.000, C 0.000 }
gfCNCPoint3[768] = {X 302.7148, Y 86.7137, Z -3.8333, A 0.000, B 0.000, C 0.000 }
gfCNCPoint3[769] = {X 302.6357, Y 84.5988, Z -3.8333, A 0.000, B 0.000, C 0.000 }
gfCNCPoint3[770] = {X 302.6368, Y 66.5621, Z -3.8333, A 0.000, B 0.000, C 0.000 }
gfCNCPoint3[771] = {X 301.5837, Y 65.6069, Z -3.8333, A 0.000, B 0.000, C 0.000 }
gfCNCPoint3[772] = {X 300.6820, Y 64.5078, Z -3.8333, A 0.000, B 0.000, C 0.000 }
gfCNCPoint3[773] = {X 298.7203, Y 63.1251, Z -3.8333, A 0.000, B 0.000, C 0.000 }
gfCNCPoint3[774] = {X 298.0342, Y 63.9596, Z -3.8333, A 0.000, B 0.000, C 0.000 }
gfCNCPoint3[775] = {X 297.2324, Y 64.6837, Z -3.8333, A 0.000, B 0.000, C 0.000 }
gfCNCPoint3[776] = {X 296.3324, Y 65.2814, Z -3.8333, A 0.000, B 0.000, C 0.000 }
gfCNCPoint3[777] = {X 296.3324, Y 90.7166, Z -3.8333, A 0.000, B 0.000, C 0.000 }
gfCNCPoint3[778] = {X 297.3126, Y 91.3792, Z -3.8333, A 0.000, B 0.000, C 0.000 }
gfCNCPoint3[779] = {X 298.1731, Y 92.1912, Z -3.8333, A 0.000, B 0.000, C 0.000 }
gfCNCPoint3[780] = {X 298.8914, Y 93.1314, Z -3.8333, A 0.000, B 0.000, C 0.000 }
gfCNCPoint3[781] = {X 299.4487, Y 94.1751, Z -3.8333, A 0.000, B 0.000, C 0.000 }
gfCNCPoint3[782] = {X 299.8303, Y 95.2950, Z -3.8333, A 0.000, B 0.000, C 0.000 }
gfCNCPoint3[783] = {X 308.0992, Y 95.2950, Z -3.8333, A 0.000, B 0.000, C 0.000 }
gfCNCPoint3[784] = {X 307.0961, Y 93.7116, Z -3.8333, A 0.000, B 0.000, C 0.000 }
gfCNCPoint3[785] = {X 306.3001, Y 92.0147, Z -3.8333, A 0.000, B 0.000, C 0.000 }
gfCNCPoint3[786] = {X 305.9922, Y 91.1577, Z -3.8333, A 0.000, B 0.000, C 0.000 }
gfCNCPoint3[787] = {X 305.7373, Y 90.2835, Z -3.8333, A 0.000, B 0.000, C 0.000 }
gfCNCPoint3[788] = {X 305.3410, Y 88.4133, Z -3.8333, A 0.000, B 0.000, C 0.000 }
gfCNCPoint3[789] = {X 305.1066, Y 86.5161, Z -3.8333, A 0.000, B 0.000, C 0.000 }
gfCNCPoint3[790] = {X 305.0357, Y 84.6057, Z -3.8333, A 0.000, B 0.000, C 0.000 }
gfCNCPoint3[791] = {X 305.0368, Y 65.2846, Z -3.8333, A 0.000, B 0.000, C 0.000 }
gfCNCPoint3[792] = {X 304.1348, Y 64.6868, Z -3.8333, A 0.000, B 0.000, C 0.000 }
gfCNCPoint3[793] = {X 303.3313, Y 63.9619, Z -3.8333, A 0.000, B 0.000, C 0.000 }
gfCNCPoint3[794] = {X 302.6442, Y 63.1259, Z -3.8333, A 0.000, B 0.000, C 0.000 }
gfCNCPoint3[795] = {X 302.0792, Y 62.1785, Z -3.8333, A 0.000, B 0.000, C 0.000 }
gfCNCPoint3[796] = {X 301.6638, Y 61.1567, Z -3.8333, A 0.000, B 0.000, C 0.000 }
gfCNCPoint3[797] = {X 301.4076, Y 60.0838, Z -3.8333, A 0.000, B 0.000, C 0.000 }
gfCNCPoint3[798] = {X 301.3164, Y 58.9845, Z -3.8333, A 0.000, B 0.000, C 0.000 }
gfCNCPoint3[799] = {X 301.3162, Y 58.0000, Z -3.8333, A 0.000, B 0.000, C 0.000 }
gfCNCPoint3[800] = {X 301.4018, Y 56.8868, Z -3.8333, A 0.000, B 0.000, C 0.000 }
gfCNCPoint3[801] = {X 301.6567, Y 55.7997, Z -3.8333, A 0.000, B 0.000, C 0.000 }
gfCNCPoint3[802] = {X 302.0747, Y 54.7645, Z -3.8333, A 0.000, B 0.000, C 0.000 }
gfCNCPoint3[803] = {X 302.6462, Y 53.8053, Z -3.8333, A 0.000, B 0.000, C 0.000 }
gfCNCPoint3[804] = {X 303.3281, Y 52.9755, Z -3.8333, A 0.000, B 0.000, C 0.000 }
gfCNCPoint3[805] = {X 304.1247, Y 52.2551, Z -3.8333, A 0.000, B 0.000, C 0.000 }
gfCNCPoint3[806] = {X 305.0187, Y 51.6597, Z -3.8333, A 0.000, B 0.000, C 0.000 }
gfCNCPoint3[807] = {X 306.1514, Y 51.1428, Z -3.8333, A 0.000, B 0.000, C 0.000 }
gfCNCPoint3[808] = {X 307.3557, Y 50.8265, Z -3.8333, A 0.000, B 0.000, C 0.000 }
gfCNCPoint3[809] = {X 308.5962, Y 50.7200, Z -3.8333, A 0.000, B 0.000, C 0.000 }
gfCNCPoint3[810] = {X 324.3107, Y 50.7200, Z -3.8333, A 0.000, B 0.000, C 0.000 }
gfCNCPoint3[811] = {X 325.2469, Y 50.7804, Z -3.8333, A 0.000, B 0.000, C 0.000 }
gfCNCPoint3[812] = {X 326.1675, Y 50.9608, Z -3.8333, A 0.000, B 0.000, C 0.000 }
gfCNCPoint3[813] = {X 326.5260, Y 51.0653, Z -3.8333, A 0.000, B 0.000, C 0.000 }
gfCNCPoint3[814] = {X 326.8787, Y 51.1880, Z -3.8333, A 0.000, B 0.000, C 0.000 }
gfCNCPoint3[815] = {X 327.4511, Y 51.4322, Z -3.8333, A 0.000, B 0.000, C 0.000 }
gfCNCPoint3[816] = {X 328.0006, Y 51.7244, Z -3.8333, A 0.000, B 0.000, C 0.000 }
gfCNCPoint3[817] = {X 328.5423, Y 52.0761, Z -3.8333, A 0.000, B 0.000, C 0.000 }
gfCNCPoint3[818] = {X 329.0506, Y 52.4745, Z -3.8333, A 0.000, B 0.000, C 0.000 }
gfCNCPoint3[819] = {X 329.9280, Y 53.3692, Z -3.8333, A 0.000, B 0.000, C 0.000 }
gfCNCPoint3[820] = {X 330.6390, Y 54.4012, Z -3.8333, A 0.000, B 0.000, C 0.000 }
gfCNCPoint3[821] = {X 331.1624, Y 55.5399, Z -3.8333, A 0.000, B 0.000, C 0.000 }
gfCNCPoint3[822] = {X 331.4828, Y 56.7515, Z -3.8333, A 0.000, B 0.000, C 0.000 }
gfCNCPoint3[823] = {X 331.5907, Y 58.0000, Z -3.8333, A 0.000, B 0.000, C 0.000 }
gfCNCPoint3[824] = {X 331.5907, Y 58.9456, Z -3.8333, A 0.000, B 0.000, C 0.000 }
gfCNCPoint3[825] = {X 331.4723, Y 60.2215, Z -3.8333, A 0.000, B 0.000, C 0.000 }
gfCNCPoint3[826] = {X 331.1333, Y 61.4572, Z -3.8333, A 0.000, B 0.000, C 0.000 }
gfCNCPoint3[827] = {X 330.5840, Y 62.6148, Z -3.8333, A 0.000, B 0.000, C 0.000 }
gfCNCPoint3[828] = {X 329.8412, Y 63.6589, Z -3.8333, A 0.000, B 0.000, C 0.000 }
gfCNCPoint3[829] = {X 328.9277, Y 64.5575, Z -3.8333, A 0.000, B 0.000, C 0.000 }
gfCNCPoint3[830] = {X 327.8715, Y 65.2829, Z -3.8333, A 0.000, B 0.000, C 0.000 }
gfCNCPoint3[831] = {X 327.8729, Y 83.2150, Z -3.8333, A 0.000, B 0.000, C 0.000 }
gfCNCPoint3[832] = {X 327.8864, Y 84.5920, Z -3.8333, A 0.000, B 0.000, C 0.000 }
gfCNCPoint3[833] = {X 327.8958, Y 84.9543, Z -3.8333, A 0.000, B 0.000, C 0.000 }
gfCNCPoint3[834] = {X 327.9226, Y 85.3157, Z -3.8333, A 0.000, B 0.000, C 0.000 }
gfCNCPoint3[835] = {X 328.8643, Y 85.6731, Z -3.8333, A 0.000, B 0.000, C 0.000 }
gfCNCPoint3[836] = {X 329.8341, Y 85.9448, Z -3.8333, A 0.000, B 0.000, C 0.000 }
gfCNCPoint3[837] = {X 332.7078, Y 86.5206, Z -3.8333, A 0.000, B 0.000, C 0.000 }
gfCNCPoint3[838] = {X 335.6156, Y 86.8874, Z -3.8333, A 0.000, B 0.000, C 0.000 }
gfCNCPoint3[839] = {X 339.6625, Y 87.2007, Z -3.8333, A 0.000, B 0.000, C 0.000 }
gfCNCPoint3[840] = {X 343.7178, Y 87.3762, Z -3.8333, A 0.000, B 0.000, C 0.000 }
gfCNCPoint3[841] = {X 347.7767, Y 87.4136, Z -3.8333, A 0.000, B 0.000, C 0.000 }
gfCNCPoint3[842] = {X 352.0643, Y 87.3769, Z -3.8333, A 0.000, B 0.000, C 0.000 }
gfCNCPoint3[843] = {X 356.3478, Y 87.1857, Z -3.8333, A 0.000, B 0.000, C 0.000 }
gfCNCPoint3[844] = {X 360.6216, Y 86.8402, Z -3.8333, A 0.000, B 0.000, C 0.000 }
gfCNCPoint3[845] = {X 362.7646, Y 86.5740, Z -3.8333, A 0.000, B 0.000, C 0.000 }
gfCNCPoint3[846] = {X 364.8876, Y 86.1792, Z -3.8333, A 0.000, B 0.000, C 0.000 }
gfCNCPoint3[847] = {X 366.9831, Y 85.6572, Z -3.8333, A 0.000, B 0.000, C 0.000 }
gfCNCPoint3[848] = {X 367.4430, Y 85.5109, Z -3.8333, A 0.000, B 0.000, C 0.000 }
gfCNCPoint3[849] = {X 367.8892, Y 85.3267, Z -3.8333, A 0.000, B 0.000, C 0.000 }
gfCNCPoint3[850] = {X 367.9426, Y 84.5784, Z -3.8333, A 0.000, B 0.000, C 0.000 }
gfCNCPoint3[851] = {X 367.9604, Y 83.8284, Z -3.8333, A 0.000, B 0.000, C 0.000 }
gfCNCPoint3[852] = {X 367.9590, Y 65.2841, Z -3.8333, A 0.000, B 0.000, C 0.000 }
gfCNCPoint3[853] = {X 366.9051, Y 64.5650, Z -3.8333, A 0.000, B 0.000, C 0.000 }
gfCNCPoint3[854] = {X 365.9929, Y 63.6730, Z -3.8333, A 0.000, B 0.000, C 0.000 }
gfCNCPoint3[855] = {X 365.2505, Y 62.6355, Z -3.8333, A 0.000, B 0.000, C 0.000 }
gfCNCPoint3[856] = {X 364.7005, Y 61.4842, Z -3.8333, A 0.000, B 0.000, C 0.000 }
gfCNCPoint3[857] = {X 364.3601, Y 60.2546, Z -3.8333, A 0.000, B 0.000, C 0.000 }
gfCNCPoint3[858] = {X 364.2395, Y 58.9845, Z -3.8333, A 0.000, B 0.000, C 0.000 }
gfCNCPoint3[859] = {X 364.2393, Y 58.0000, Z -3.8333, A 0.000, B 0.000, C 0.000 }
gfCNCPoint3[860] = {X 364.3499, Y 56.7358, Z -3.8333, A 0.000, B 0.000, C 0.000 }
gfCNCPoint3[861] = {X 364.6783, Y 55.5101, Z -3.8333, A 0.000, B 0.000, C 0.000 }
gfCNCPoint3[862] = {X 365.2146, Y 54.3600, Z -3.8333, A 0.000, B 0.000, C 0.000 }
gfCNCPoint3[863] = {X 365.9425, Y 53.3205, Z -3.8333, A 0.000, B 0.000, C 0.000 }
gfCNCPoint3[864] = {X 366.8398, Y 52.4232, Z -3.8333, A 0.000, B 0.000, C 0.000 }
gfCNCPoint3[865] = {X 367.8793, Y 51.6953, Z -3.8333, A 0.000, B 0.000, C 0.000 }
gfCNCPoint3[866] = {X 369.0294, Y 51.1590, Z -3.8333, A 0.000, B 0.000, C 0.000 }
gfCNCPoint3[867] = {X 370.2551, Y 50.8306, Z -3.8333, A 0.000, B 0.000, C 0.000 }
gfCNCPoint3[868] = {X 371.5193, Y 50.7200, Z -3.8333, A 0.000, B 0.000, C 0.000 }
gfCNCPoint3[869] = {X 388.0597, Y 50.7200, Z -3.8333, A 0.000, B 0.000, C 0.000 }
gfCNCPoint3[870] = {X 389.2271, Y 50.8142, Z -3.8333, A 0.000, B 0.000, C 0.000 }
gfCNCPoint3[871] = {X 390.3643, Y 51.0944, Z -3.8333, A 0.000, B 0.000, C 0.000 }
gfCNCPoint3[872] = {X 391.4418, Y 51.5533, Z -3.8333, A 0.000, B 0.000, C 0.000 }
gfCNCPoint3[873] = {X 392.4319, Y 52.1791, Z -3.8333, A 0.000, B 0.000, C 0.000 }
gfCNCPoint3[874] = {X 393.3087, Y 52.9556, Z -3.8333, A 0.000, B 0.000, C 0.000 }
gfCNCPoint3[875] = {X 394.1855, Y 52.1791, Z -3.8333, A 0.000, B 0.000, C 0.000 }
gfCNCPoint3[876] = {X 395.1756, Y 51.5533, Z -3.8333, A 0.000, B 0.000, C 0.000 }
gfCNCPoint3[877] = {X 396.2531, Y 51.0944, Z -3.8333, A 0.000, B 0.000, C 0.000 }
gfCNCPoint3[878] = {X 397.3903, Y 50.8142, Z -3.8333, A 0.000, B 0.000, C 0.000 }
gfCNCPoint3[879] = {X 398.5577, Y 50.7200, Z -3.8333, A 0.000, B 0.000, C 0.000 }
gfCNCPoint3[880] = {X 419.4886, Y 50.7200, Z -3.8333, A 0.000, B 0.000, C 0.000 }
gfCNCPoint3[881] = {X 420.6740, Y 50.8172, Z -3.8333, A 0.000, B 0.000, C 0.000 }
gfCNCPoint3[882] = {X 421.8277, Y 51.1060, Z -3.8333, A 0.000, B 0.000, C 0.000 }
gfCNCPoint3[883] = {X 422.9190, Y 51.5789, Z -3.8333, A 0.000, B 0.000, C 0.000 }
gfCNCPoint3[884] = {X 423.9188, Y 52.2232, Z -3.8333, A 0.000, B 0.000, C 0.000 }
gfCNCPoint3[885] = {X 424.8003, Y 53.0216, Z -3.8333, A 0.000, B 0.000, C 0.000 }
gfCNCPoint3[886] = {X 425.5400, Y 53.9530, Z -3.8333, A 0.000, B 0.000, C 0.000 }
gfCNCPoint3[887] = {X 426.1182, Y 54.9923, Z -3.8333, A 0.000, B 0.000, C 0.000 }
gfCNCPoint3[888] = {X 426.5195, Y 56.1119, Z -3.8333, A 0.000, B 0.000, C 0.000 }
gfCNCPoint3[889] = {X 430.7007, Y 57.7414, Z -3.8333, A 0.000, B 0.000, C 0.000 }
gfCNCPoint3[890] = {X 454.8990, Y 67.3421, Z -3.8333, A 0.000, B 0.000, C 0.000 }
gfCNCPoint3[891] = {X 454.8992, Y 65.2840, Z -3.8333, A 0.000, B 0.000, C 0.000 }
gfCNCPoint3[892] = {X 453.8919, Y 64.6028, Z -3.8333, A 0.000, B 0.000, C 0.000 }
gfCNCPoint3[893] = {X 453.0120, Y 63.7634, Z -3.8333, A 0.000, B 0.000, C 0.000 }
gfCNCPoint3[894] = {X 452.2842, Y 62.7892, Z -3.8333, A 0.000, B 0.000, C 0.000 }
gfCNCPoint3[895] = {X 451.7286, Y 61.7075, Z -3.8333, A 0.000, B 0.000, C 0.000 }
gfCNCPoint3[896] = {X 451.4297, Y 60.8258, Z -3.8333, A 0.000, B 0.000, C 0.000 }
gfCNCPoint3[897] = {X 451.2457, Y 59.9132, Z -3.8333, A 0.000, B 0.000, C 0.000 }
gfCNCPoint3[898] = {X 451.1798, Y 58.9845, Z -3.8333, A 0.000, B 0.000, C 0.000 }
gfCNCPoint3[899] = {X 451.1796, Y 58.0000, Z -3.8333, A 0.000, B 0.000, C 0.000 }
gfCNCPoint3[900] = {X 451.2795, Y 56.7981, Z -3.8333, A 0.000, B 0.000, C 0.000 }
gfCNCPoint3[901] = {X 451.5765, Y 55.6291, Z -3.8333, A 0.000, B 0.000, C 0.000 }
gfCNCPoint3[902] = {X 452.0624, Y 54.5253, Z -3.8333, A 0.000, B 0.000, C 0.000 }
gfCNCPoint3[903] = {X 452.7238, Y 53.5168, Z -3.8333, A 0.000, B 0.000, C 0.000 }
gfCNCPoint3[904] = {X 453.5427, Y 52.6313, Z -3.8333, A 0.000, B 0.000, C 0.000 }
gfCNCPoint3[905] = {X 454.4966, Y 51.8932, Z -3.8333, A 0.000, B 0.000, C 0.000 }
gfCNCPoint3[906] = {X 455.4133, Y 51.3880, Z -3.8333, A 0.000, B 0.000, C 0.000 }
gfCNCPoint3[907] = {X 456.3931, Y 51.0195, Z -3.8333, A 0.000, B 0.000, C 0.000 }
gfCNCPoint3[908] = {X 457.4155, Y 50.7953, Z -3.8333, A 0.000, B 0.000, C 0.000 }
gfCNCPoint3[909] = {X 458.4596, Y 50.7200, Z -3.8333, A 0.000, B 0.000, C 0.000 }
gfCNCPoint3[910] = {X 475.0000, Y 50.7200, Z -3.8333, A 0.000, B 0.000, C 0.000 }
gfCNCPoint3[911] = {X 476.0441, Y 50.7953, Z -3.8333, A 0.000, B 0.000, C 0.000 }
gfCNCPoint3[912] = {X 477.0665, Y 51.0195, Z -3.8333, A 0.000, B 0.000, C 0.000 }
gfCNCPoint3[913] = {X 478.0463, Y 51.3880, Z -3.8333, A 0.000, B 0.000, C 0.000 }
gfCNCPoint3[914] = {X 478.9630, Y 51.8932, Z -3.8333, A 0.000, B 0.000, C 0.000 }
gfCNCPoint3[915] = {X 479.9169, Y 52.6313, Z -3.8333, A 0.000, B 0.000, C 0.000 }
gfCNCPoint3[916] = {X 480.7358, Y 53.5168, Z -3.8333, A 0.000, B 0.000, C 0.000 }
gfCNCPoint3[917] = {X 481.3972, Y 54.5253, Z -3.8333, A 0.000, B 0.000, C 0.000 }
gfCNCPoint3[918] = {X 481.8831, Y 55.6291, Z -3.8333, A 0.000, B 0.000, C 0.000 }
gfCNCPoint3[919] = {X 482.1801, Y 56.7981, Z -3.8333, A 0.000, B 0.000, C 0.000 }
gfCNCPoint3[920] = {X 482.2800, Y 58.0000, Z -3.8333, A 0.000, B 0.000, C 0.000 }
gfCNCPoint3[921] = {X 482.2798, Y 58.9942, Z -3.8333, A 0.000, B 0.000, C 0.000 }
gfCNCPoint3[922] = {X 482.1577, Y 60.2626, Z -3.8333, A 0.000, B 0.000, C 0.000 }
gfCNCPoint3[923] = {X 481.8164, Y 61.4904, Z -3.8333, A 0.000, B 0.000, C 0.000 }
gfCNCPoint3[924] = {X 481.2663, Y 62.6398, Z -3.8333, A 0.000, B 0.000, C 0.000 }
gfCNCPoint3[925] = {X 480.5241, Y 63.6756, Z -3.8333, A 0.000, B 0.000, C 0.000 }
gfCNCPoint3[926] = {X 479.6127, Y 64.5662, Z -3.8333, A 0.000, B 0.000, C 0.000 }
gfCNCPoint3[927] = {X 478.5600, Y 65.2842, Z -3.8333, A 0.000, B 0.000, C 0.000 }
gfCNCPoint3[928] = {X 478.5604, Y 90.7245, Z -3.8333, A 0.000, B 0.000, C 0.000 }
gfCNCPoint3[929] = {X 479.5429, Y 91.3831, Z -3.8333, A 0.000, B 0.000, C 0.000 }
gfCNCPoint3[930] = {X 480.4054, Y 92.1926, Z -3.8333, A 0.000, B 0.000, C 0.000 }
gfCNCPoint3[931] = {X 481.1248, Y 93.1316, Z -3.8333, A 0.000, B 0.000, C 0.000 }
gfCNCPoint3[932] = {X 481.6820, Y 94.1749, Z -3.8333, A 0.000, B 0.000, C 0.000 }
gfCNCPoint3[933] = {X 482.0623, Y 95.2950, Z -3.8333, A 0.000, B 0.000, C 0.000 }
gfCNCPoint3[934] = {X 507.6816, Y 95.2950, Z -3.8333, A 0.000, B 0.000, C 0.000 }
gfCNCPoint3[935] = {X 507.6816, Y 97.6950, Z -3.8333, A 0.000, B 0.000, C 0.000 }
gfCNCPoint3[936] = {X 597.6965, Y 97.6950, Z -3.8333, A 0.000, B 0.000, C 0.000 }
gfCNCPoint3[937] = {X 597.6965, Y 51.8000, Z -3.8333, A 0.000, B 0.000, C 0.000 }
gfCNCPoint3[938] = {X 593.5565, Y 51.8000, Z -3.8333, A 0.000, B 0.000, C 0.000 }
gfCNCPoint3[939] = {X 592.3428, Y 51.6908, Z -3.8333, A 0.000, B 0.000, C 0.000 }
gfCNCPoint3[940] = {X 591.1680, Y 51.3667, Z -3.8333, A 0.000, B 0.000, C 0.000 }
gfCNCPoint3[941] = {X 590.0699, Y 50.8381, Z -3.8333, A 0.000, B 0.000, C 0.000 }
gfCNCPoint3[942] = {X 589.0838, Y 50.1220, Z -3.8333, A 0.000, B 0.000, C 0.000 }
gfCNCPoint3[943] = {X 588.4736, Y 49.5171, Z -3.8333, A 0.000, B 0.000, C 0.000 }
gfCNCPoint3[944] = {X 587.9446, Y 48.8401, Z -3.8333, A 0.000, B 0.000, C 0.000 }
gfCNCPoint3[945] = {X 587.5052, Y 48.1018, Z -3.8333, A 0.000, B 0.000, C 0.000 }
gfCNCPoint3[946] = {X 587.1971, Y 48.6407, Z -3.8333, A 0.000, B 0.000, C 0.000 }
gfCNCPoint3[947] = {X 586.8412, Y 49.1493, Z -3.8333, A 0.000, B 0.000, C 0.000 }
gfCNCPoint3[948] = {X 586.4078, Y 49.6581, Z -3.8333, A 0.000, B 0.000, C 0.000 }
gfCNCPoint3[949] = {X 585.9266, Y 50.1220, Z -3.8333, A 0.000, B 0.000, C 0.000 }
gfCNCPoint3[950] = {X 585.1803, Y 50.6880, Z -3.8333, A 0.000, B 0.000, C 0.000 }
gfCNCPoint3[951] = {X 584.3634, Y 51.1461, Z -3.8333, A 0.000, B 0.000, C 0.000 }
gfCNCPoint3[952] = {X 583.3013, Y 51.5442, Z -3.8333, A 0.000, B 0.000, C 0.000 }
gfCNCPoint3[953] = {X 582.1877, Y 51.7603, Z -3.8333, A 0.000, B 0.000, C 0.000 }
gfCNCPoint3[954] = {X 581.0538, Y 51.7882, Z -3.8333, A 0.000, B 0.000, C 0.000 }
gfCNCPoint3[955] = {X 579.9310, Y 51.6273, Z -3.8333, A 0.000, B 0.000, C 0.000 }
gfCNCPoint3[956] = {X 578.8505, Y 51.2819, Z -3.8333, A 0.000, B 0.000, C 0.000 }
gfCNCPoint3[957] = {X 577.8425, Y 50.7618, Z -3.8333, A 0.000, B 0.000, C 0.000 }
gfCNCPoint3[958] = {X 576.9350, Y 50.0813, Z -3.8333, A 0.000, B 0.000, C 0.000 }
gfCNCPoint3[959] = {X 576.3133, Y 49.4513, Z -3.8333, A 0.000, B 0.000, C 0.000 }
gfCNCPoint3[960] = {X 575.7786, Y 48.7459, Z -3.8333, A 0.000, B 0.000, C 0.000 }
gfCNCPoint3[961] = {X 575.3401, Y 47.9770, Z -3.8333, A 0.000, B 0.000, C 0.000 }
gfCNCPoint3[962] = {X 574.9017, Y 48.7459, Z -3.8333, A 0.000, B 0.000, C 0.000 }
gfCNCPoint3[963] = {X 574.3670, Y 49.4513, Z -3.8333, A 0.000, B 0.000, C 0.000 }
gfCNCPoint3[964] = {X 573.7453, Y 50.0813, Z -3.8333, A 0.000, B 0.000, C 0.000 }
gfCNCPoint3[965] = {X 572.7526, Y 50.8143, Z -3.8333, A 0.000, B 0.000, C 0.000 }
gfCNCPoint3[966] = {X 571.6437, Y 51.3558, Z -3.8333, A 0.000, B 0.000, C 0.000 }
gfCNCPoint3[967] = {X 570.4553, Y 51.6880, Z -3.8333, A 0.000, B 0.000, C 0.000 }
gfCNCPoint3[968] = {X 569.2264, Y 51.8000, Z -3.8333, A 0.000, B 0.000, C 0.000 }
gfCNCPoint3[969] = {X 562.4443, Y 51.8000, Z -3.8333, A 0.000, B 0.000, C 0.000 }
gfCNCPoint3[970] = {X 561.2635, Y 51.6967, Z -3.8333, A 0.000, B 0.000, C 0.000 }
gfCNCPoint3[971] = {X 560.1186, Y 51.3899, Z -3.8333, A 0.000, B 0.000, C 0.000 }
gfCNCPoint3[972] = {X 559.0443, Y 50.8890, Z -3.8333, A 0.000, B 0.000, C 0.000 }
gfCNCPoint3[973] = {X 558.0733, Y 50.2091, Z -3.8333, A 0.000, B 0.000, C 0.000 }
gfCNCPoint3[974] = {X 557.2352, Y 49.3710, Z -3.8333, A 0.000, B 0.000, C 0.000 }
gfCNCPoint3[975] = {X 556.5553, Y 48.4000, Z -3.8333, A 0.000, B 0.000, C 0.000 }
gfCNCPoint3[976] = {X 556.0544, Y 47.3257, Z -3.8333, A 0.000, B 0.000, C 0.000 }
gfCNCPoint3[977] = {X 555.7476, Y 46.1808, Z -3.8333, A 0.000, B 0.000, C 0.000 }
gfCNCPoint3[978] = {X 555.6443, Y 45.0000, Z -3.8333, A 0.000, B 0.000, C 0.000 }
gfCNCPoint3[979] = {X 555.6443, Y 44.0535, Z -3.8333, A 0.000, B 0.000, C 0.000 }
gfCNCPoint3[980] = {X 555.7471, Y 42.9021, Z -3.8333, A 0.000, B 0.000, C 0.000 }
gfCNCPoint3[981] = {X 556.0426, Y 41.7844, Z -3.8333, A 0.000, B 0.000, C 0.000 }
gfCNCPoint3[982] = {X 556.5221, Y 40.7325, Z -3.8333, A 0.000, B 0.000, C 0.000 }
gfCNCPoint3[983] = {X 557.1721, Y 39.7765, Z -3.8333, A 0.000, B 0.000, C 0.000 }
gfCNCPoint3[984] = {X 557.1721, Y 10.2287, Z -3.8333, A 0.000, B 0.000, C 0.000 }
gfCNCPoint3[985] = {X 556.5258, Y 9.2825, Z -3.8333, A 0.000, B 0.000, C 0.000 }
gfCNCPoint3[986] = {X 556.0476, Y 8.2412, Z -3.8333, A 0.000, B 0.000, C 0.000 }
gfCNCPoint3[987] = {X 555.7511, Y 7.1344, Z -3.8333, A 0.000, B 0.000, C 0.000 }
gfCNCPoint3[988] = {X 555.6446, Y 5.9935, Z -3.8333, A 0.000, B 0.000, C 0.000 }
gfCNCPoint3[989] = {X 555.6443, Y 5.0000, Z -3.8333, A 0.000, B 0.000, C 0.000 }
gfCNCPoint3[990] = {X 555.6452, Y 4.8910, Z -3.8333, A 0.000, B 0.000, C 0.000 }
gfCNCPoint3[991] = {X 555.6478, Y 4.7820, Z -3.8333, A 0.000, B 0.000, C 0.000 }
gfCNCPoint3[992] = {X 555.8079, Y 3.5174, Z -3.8333, A 0.000, B 0.000, C 0.000 }
gfCNCPoint3[993] = {X 556.2011, Y 2.3050, Z -3.8333, A 0.000, B 0.000, C 0.000 }
gfCNCPoint3[994] = {X 358.2587, Y 2.3050, Z -3.8333, A 0.000, B 0.000, C 0.000 }
gfCNCPoint3[995] = {X 360.1201, Y 3.4746, Z -3.8333, A 0.000, B 0.000, C 0.000 }
gfCNCPoint3[996] = {X 361.8529, Y 4.8276, Z -3.8333, A 0.000, B 0.000, C 0.000 }
gfCNCPoint3[997] = {X 363.4390, Y 6.3497, Z -3.8333, A 0.000, B 0.000, C 0.000 }
gfCNCPoint3[998] = {X 363.7850, Y 6.7263, Z -3.8333, A 0.000, B 0.000, C 0.000 }
gfCNCPoint3[999] = {X 364.1220, Y 7.1109, Z -3.8333, A 0.000, B 0.000, C 0.000 }
gfCNCPoint3[1000] = {X 365.6210, Y 9.0455, Z -3.8333, A 0.000, B 0.000, C 0.000 }
gfCNCPoint3[1001] = {X 366.9260, Y 11.1160, Z -3.8333, A 0.000, B 0.000, C 0.000 }
gfCNCPoint3[1002] = {X 368.0245, Y 13.3030, Z -3.8333, A 0.000, B 0.000, C 0.000 }
gfCNCPoint3[1003] = {X 368.9064, Y 15.5860, Z -3.8333, A 0.000, B 0.000, C 0.000 }
gfCNCPoint3[1004] = {X 369.5634, Y 17.9436, Z -3.8333, A 0.000, B 0.000, C 0.000 }
gfCNCPoint3[1005] = {X 370.0543, Y 20.6266, Z -3.8333, A 0.000, B 0.000, C 0.000 }
gfCNCPoint3[1006] = {X 370.3162, Y 23.3416, Z -3.8333, A 0.000, B 0.000, C 0.000 }
gfCNCPoint3[1007] = {X 370.3472, Y 26.0690, Z -3.8333, A 0.000, B 0.000, C 0.000 }
gfCNCPoint3[1008] = {X 370.1472, Y 28.7892, Z -3.8333, A 0.000, B 0.000, C 0.000 }
gfCNCPoint3[1009] = {X 369.7174, Y 31.4828, Z -3.8333, A 0.000, B 0.000, C 0.000 }
gfCNCPoint3[1010] = {X 369.1818, Y 33.6343, Z -3.8333, A 0.000, B 0.000, C 0.000 }
gfCNCPoint3[1011] = {X 368.4582, Y 35.7302, Z -3.8333, A 0.000, B 0.000, C 0.000 }
gfCNCPoint3[1012] = {X 367.5523, Y 37.7540, Z -3.8333, A 0.000, B 0.000, C 0.000 }
gfCNCPoint3[1013] = {X 366.4713, Y 39.6898, Z -3.8333, A 0.000, B 0.000, C 0.000 }
gfCNCPoint3[1014] = {X 365.2235, Y 41.5226, Z -3.8333, A 0.000, B 0.000, C 0.000 }
gfCNCPoint3[1015] = {X 365.0833, Y 41.7127, Z -3.8333, A 0.000, B 0.000, C 0.000 }
gfCNCPoint3[1016] = {X 364.4574, Y 42.4812, Z -3.8333, A 0.000, B 0.000, C 0.000 }
gfCNCPoint3[1017] = {X 363.1634, Y 43.9329, Z -3.8333, A 0.000, B 0.000, C 0.000 }
gfCNCPoint3[1018] = {X 361.7455, Y 45.2639, Z -3.8333, A 0.000, B 0.000, C 0.000 }
gfCNCPoint3[1019] = {X 360.2149, Y 46.4635, Z -3.8333, A 0.000, B 0.000, C 0.000 }
gfCNCPoint3[1020] = {X 358.5837, Y 47.5223, Z -3.8333, A 0.000, B 0.000, C 0.000 }
gfCNCPoint3[1021] = {X 356.8649, Y 48.4319, Z -3.8333, A 0.000, B 0.000, C 0.000 }
gfCNCPoint3[1022] = {X 356.4678, Y 48.6199, Z -3.8333, A 0.000, B 0.000, C 0.000 }
gfCNCPoint3[1023] = {X 354.6708, Y 49.3140, Z -3.8333, A 0.000, B 0.000, C 0.000 }
gfCNCPoint3[1024] = {X 352.8232, Y 49.8590, Z -3.8333, A 0.000, B 0.000, C 0.000 }
gfCNCPoint3[1025] = {X 350.9372, Y 50.2513, Z -3.8333, A 0.000, B 0.000, C 0.000 }
gfCNCPoint3[1026] = {X 349.0255, Y 50.4884, Z -3.8333, A 0.000, B 0.000, C 0.000 }
gfCNCPoint3[1027] = {X 347.1008, Y 50.5686, Z -3.8333, A 0.000, B 0.000, C 0.000 }
gfCNCPoint3[1028] = {X 344.9874, Y 50.5324, Z -3.8333, A 0.000, B 0.000, C 0.000 }
gfCNCPoint3[1029] = {X 342.8850, Y 50.3132, Z -3.8333, A 0.000, B 0.000, C 0.000 }
gfCNCPoint3[1030] = {X 340.8096, Y 49.9126, Z -3.8333, A 0.000, B 0.000, C 0.000 }
gfCNCPoint3[1031] = {X 338.7767, Y 49.3337, Z -3.8333, A 0.000, B 0.000, C 0.000 }
gfCNCPoint3[1032] = {X 336.8016, Y 48.5808, Z -3.8333, A 0.000, B 0.000, C 0.000 }
gfCNCPoint3[1033] = {X 334.8991, Y 47.6595, Z -3.8333, A 0.000, B 0.000, C 0.000 }
gfCNCPoint3[1034] = {X 333.3419, Y 46.7032, Z -3.8333, A 0.000, B 0.000, C 0.000 }
gfCNCPoint3[1035] = {X 331.8607, Y 45.6331, Z -3.8333, A 0.000, B 0.000, C 0.000 }
gfCNCPoint3[1036] = {X 330.4638, Y 44.4550, Z -3.8333, A 0.000, B 0.000, C 0.000 }
gfCNCPoint3[1037] = {X 329.4665, Y 44.4078, Z -3.8333, A 0.000, B 0.000, C 0.000 }
gfCNCPoint3[1038] = {X 328.4997, Y 44.1587, Z -3.8333, A 0.000, B 0.000, C 0.000 }
gfCNCPoint3[1039] = {X 327.6038, Y 43.7181, Z -3.8333, A 0.000, B 0.000, C 0.000 }
gfCNCPoint3[1040] = {X 326.8164, Y 43.1044, Z -3.8333, A 0.000, B 0.000, C 0.000 }
gfCNCPoint3[1041] = {X 326.1897, Y 42.4934, Z -3.8333, A 0.000, B 0.000, C 0.000 }
gfCNCPoint3[1042] = {X 325.5686, Y 41.7541, Z -3.8333, A 0.000, B 0.000, C 0.000 }
gfCNCPoint3[1043] = {X 325.1052, Y 40.9070, Z -3.8333, A 0.000, B 0.000, C 0.000 }
gfCNCPoint3[1044] = {X 324.8177, Y 39.9852, Z -3.8333, A 0.000, B 0.000, C 0.000 }
gfCNCPoint3[1045] = {X 324.7172, Y 39.0249, Z -3.8333, A 0.000, B 0.000, C 0.000 }
gfCNCPoint3[1046] = {X 324.8079, Y 38.0635, Z -3.8333, A 0.000, B 0.000, C 0.000 }
gfCNCPoint3[1047] = {X 325.0860, Y 37.1389, Z -3.8333, A 0.000, B 0.000, C 0.000 }
gfCNCPoint3[1048] = {X 325.5408, Y 36.2871, Z -3.8333, A 0.000, B 0.000, C 0.000 }
gfCNCPoint3[1049] = {X 329.7765, Y 29.9537, Z -3.8333, A 0.000, B 0.000, C 0.000 }
gfCNCPoint3[1050] = {X 330.4614, Y 29.1399, Z -3.8333, A 0.000, B 0.000, C 0.000 }
gfCNCPoint3[1051] = {X 331.3063, Y 28.4938, Z -3.8333, A 0.000, B 0.000, C 0.000 }
gfCNCPoint3[1052] = {X 332.2712, Y 28.0462, Z -3.8333, A 0.000, B 0.000, C 0.000 }
gfCNCPoint3[1053] = {X 333.3101, Y 27.8182, Z -3.8333, A 0.000, B 0.000, C 0.000 }
gfCNCPoint3[1054] = {X 334.3737, Y 27.8207, Z -3.8333, A 0.000, B 0.000, C 0.000 }
gfCNCPoint3[1055] = {X 335.4116, Y 28.0536, Z -3.8333, A 0.000, B 0.000, C 0.000 }
gfCNCPoint3[1056] = {X 336.3743, Y 28.5058, Z -3.8333, A 0.000, B 0.000, C 0.000 }
gfCNCPoint3[1057] = {X 337.2162, Y 29.1559, Z -3.8333, A 0.000, B 0.000, C 0.000 }
gfCNCPoint3[1058] = {X 337.8209, Y 29.7387, Z -3.8333, A 0.000, B 0.000, C 0.000 }
gfCNCPoint3[1059] = {X 338.4997, Y 30.5716, Z -3.8333, A 0.000, B 0.000, C 0.000 }
gfCNCPoint3[1060] = {X 338.9799, Y 31.5328, Z -3.8333, A 0.000, B 0.000, C 0.000 }
gfCNCPoint3[1061] = {X 339.2381, Y 32.5758, Z -3.8333, A 0.000, B 0.000, C 0.000 }
gfCNCPoint3[1062] = {X 339.2618, Y 33.6500, Z -3.8333, A 0.000, B 0.000, C 0.000 }
gfCNCPoint3[1063] = {X 339.9065, Y 34.2215, Z -3.8333, A 0.000, B 0.000, C 0.000 }
gfCNCPoint3[1064] = {X 340.5754, Y 34.7646, Z -3.8333, A 0.000, B 0.000, C 0.000 }
gfCNCPoint3[1065] = {X 341.8072, Y 35.5731, Z -3.8333, A 0.000, B 0.000, C 0.000 }
gfCNCPoint3[1066] = {X 343.1439, Y 36.1930, Z -3.8333, A 0.000, B 0.000, C 0.000 }
gfCNCPoint3[1067] = {X 344.5568, Y 36.6108, Z -3.8333, A 0.000, B 0.000, C 0.000 }
gfCNCPoint3[1068] = {X 346.0157, Y 36.8177, Z -3.8333, A 0.000, B 0.000, C 0.000 }
gfCNCPoint3[1069] = {X 347.4891, Y 36.8092, Z -3.8333, A 0.000, B 0.000, C 0.000 }
gfCNCPoint3[1070] = {X 348.8384, Y 36.6281, Z -3.8333, A 0.000, B 0.000, C 0.000 }
gfCNCPoint3[1071] = {X 350.1402, Y 36.2297, Z -3.8333, A 0.000, B 0.000, C 0.000 }
gfCNCPoint3[1072] = {X 351.3599, Y 35.6247, Z -3.8333, A 0.000, B 0.000, C 0.000 }
gfCNCPoint3[1073] = {X 352.4648, Y 34.8292, Z -3.8333, A 0.000, B 0.000, C 0.000 }
gfCNCPoint3[1074] = {X 353.5662, Y 33.7594, Z -3.8333, A 0.000, B 0.000, C 0.000 }
gfCNCPoint3[1075] = {X 354.5195, Y 32.5557, Z -3.8333, A 0.000, B 0.000, C 0.000 }
gfCNCPoint3[1076] = {X 355.3084, Y 31.2383, Z -3.8333, A 0.000, B 0.000, C 0.000 }
gfCNCPoint3[1077] = {X 355.9197, Y 29.8297, Z -3.8333, A 0.000, B 0.000, C 0.000 }
gfCNCPoint3[1078] = {X 356.3429, Y 28.3537, Z -3.8333, A 0.000, B 0.000, C 0.000 }
gfCNCPoint3[1079] = {X 356.6075, Y 26.7186, Z -3.8333, A 0.000, B 0.000, C 0.000 }
gfCNCPoint3[1080] = {X 356.7152, Y 25.0657, Z -3.8333, A 0.000, B 0.000, C 0.000 }
gfCNCPoint3[1081] = {X 356.6651, Y 23.4100, Z -3.8333, A 0.000, B 0.000, C 0.000 }
gfCNCPoint3[1082] = {X 356.4576, Y 21.7667, Z -3.8333, A 0.000, B 0.000, C 0.000 }
gfCNCPoint3[1083] = {X 356.1373, Y 20.3836, Z -3.8333, A 0.000, B 0.000, C 0.000 }
gfCNCPoint3[1084] = {X 355.6482, Y 19.0509, Z -3.8333, A 0.000, B 0.000, C 0.000 }
gfCNCPoint3[1085] = {X 354.9977, Y 17.7891, Z -3.8333, A 0.000, B 0.000, C 0.000 }
gfCNCPoint3[1086] = {X 354.1959, Y 16.6175, Z -3.8333, A 0.000, B 0.000, C 0.000 }
gfCNCPoint3[1087] = {X 353.3638, Y 15.6891, Z -3.8333, A 0.000, B 0.000, C 0.000 }
gfCNCPoint3[1088] = {X 352.4073, Y 14.8896, Z -3.8333, A 0.000, B 0.000, C 0.000 }
gfCNCPoint3[1089] = {X 351.3460, Y 14.2353, Z -3.8333, A 0.000, B 0.000, C 0.000 }
gfCNCPoint3[1090] = {X 350.2020, Y 13.7398, Z -3.8333, A 0.000, B 0.000, C 0.000 }
gfCNCPoint3[1091] = {X 348.9988, Y 13.4134, Z -3.8333, A 0.000, B 0.000, C 0.000 }
gfCNCPoint3[1092] = {X 347.3615, Y 13.2067, Z -3.8333, A 0.000, B 0.000, C 0.000 }
gfCNCPoint3[1093] = {X 345.7113, Y 13.2120, Z -3.8333, A 0.000, B 0.000, C 0.000 }
gfCNCPoint3[1094] = {X 344.0754, Y 13.4293, Z -3.8333, A 0.000, B 0.000, C 0.000 }
gfCNCPoint3[1095] = {X 342.4810, Y 13.8548, Z -3.8333, A 0.000, B 0.000, C 0.000 }
gfCNCPoint3[1096] = {X 340.9544, Y 14.4815, Z -3.8333, A 0.000, B 0.000, C 0.000 }
gfCNCPoint3[1097] = {X 339.5210, Y 15.2992, Z -3.8333, A 0.000, B 0.000, C 0.000 }
gfCNCPoint3[1098] = {X 339.4272, Y 16.1849, Z -3.8333, A 0.000, B 0.000, C 0.000 }
gfCNCPoint3[1099] = {X 339.1741, Y 17.0390, Z -3.8333, A 0.000, B 0.000, C 0.000 }
gfCNCPoint3[1100] = {X 338.7699, Y 17.8327, Z -3.8333, A 0.000, B 0.000, C 0.000 }
gfCNCPoint3[1101] = {X 338.2282, Y 18.5398, Z -3.8333, A 0.000, B 0.000, C 0.000 }
gfCNCPoint3[1102] = {X 337.5670, Y 19.1366, Z -3.8333, A 0.000, B 0.000, C 0.000 }
gfCNCPoint3[1103] = {X 336.8400, Y 19.6716, Z -3.8333, A 0.000, B 0.000, C 0.000 }
gfCNCPoint3[1104] = {X 335.9171, Y 20.1909, Z -3.8333, A 0.000, B 0.000, C 0.000 }
gfCNCPoint3[1105] = {X 334.9039, Y 20.4988, Z -3.8333, A 0.000, B 0.000, C 0.000 }
gfCNCPoint3[1106] = {X 333.8481, Y 20.5809, Z -3.8333, A 0.000, B 0.000, C 0.000 }
gfCNCPoint3[1107] = {X 332.7995, Y 20.4334, Z -3.8333, A 0.000, B 0.000, C 0.000 }
gfCNCPoint3[1108] = {X 331.8074, Y 20.0631, Z -3.8333, A 0.000, B 0.000, C 0.000 }
gfCNCPoint3[1109] = {X 330.9186, Y 19.4875, Z -3.8333, A 0.000, B 0.000, C 0.000 }
gfCNCPoint3[1110] = {X 330.1748, Y 18.7338, Z -3.8333, A 0.000, B 0.000, C 0.000 }
gfCNCPoint3[1111] = {X 329.6111, Y 17.8373, Z -3.8333, A 0.000, B 0.000, C 0.000 }
gfCNCPoint3[1112] = {X 326.0906, Y 10.5950, Z -3.8333, A 0.000, B 0.000, C 0.000 }
gfCNCPoint3[1113] = {X 325.7555, Y 9.6856, Z -3.8333, A 0.000, B 0.000, C 0.000 }
gfCNCPoint3[1114] = {X 325.6067, Y 8.7279, Z -3.8333, A 0.000, B 0.000, C 0.000 }
gfCNCPoint3[1115] = {X 325.6502, Y 7.7597, Z -3.8333, A 0.000, B 0.000, C 0.000 }
gfCNCPoint3[1116] = {X 325.8841, Y 6.8192, Z -3.8333, A 0.000, B 0.000, C 0.000 }
gfCNCPoint3[1117] = {X 326.2993, Y 5.9434, Z -3.8333, A 0.000, B 0.000, C 0.000 }
gfCNCPoint3[1118] = {X 326.9295, Y 5.1131, Z -3.8333, A 0.000, B 0.000, C 0.000 }
gfCNCPoint3[1119] = {X 327.7216, Y 4.4356, Z -3.8333, A 0.000, B 0.000, C 0.000 }
gfCNCPoint3[1120] = {X 328.3967, Y 3.9733, Z -3.8333, A 0.000, B 0.000, C 0.000 }
gfCNCPoint3[1121] = {X 329.3295, Y 3.4828, Z -3.8333, A 0.000, B 0.000, C 0.000 }
gfCNCPoint3[1122] = {X 330.3458, Y 3.2040, Z -3.8333, A 0.000, B 0.000, C 0.000 }
gfCNCPoint3[1123] = {X 331.3983, Y 3.1499, Z -3.8333, A 0.000, B 0.000, C 0.000 }
gfCNCPoint3[1124] = {X 332.4378, Y 3.3230, Z -3.8333, A 0.000, B 0.000, C 0.000 }
gfCNCPoint3[1125] = {X 333.3752, Y 2.7964, Z -3.8333, A 0.000, B 0.000, C 0.000 }
gfCNCPoint3[1126] = {X 334.3316, Y 2.3050, Z -3.8333, A 0.000, B 0.000, C 0.000 }
gfCNCPoint3[1127] = {X 334.5430, Y 2.7360, Z -3.8333, A 0.000, B 0.000, C 0.000 }
gfCNCPoint3[1128] = {X 335.0195, Y 2.5077, Z -3.8333, A 0.000, B 0.000, C 0.000 }
gfCNCPoint3[1129] = {X 335.5002, Y 2.2883, Z -3.8333, A 0.000, B 0.000, C 0.000 }
gfCNCPoint3[1130] = {X 335.8480, Y 2.1335, Z -3.8333, A 0.000, B 0.000, C 0.000 }
gfCNCPoint3[1131] = {X 337.9512, Y 1.3130, Z -3.8333, A 0.000, B 0.000, C 0.000 }
gfCNCPoint3[1132] = {X 340.1168, Y 0.6754, Z -3.8333, A 0.000, B 0.000, C 0.000 }
gfCNCPoint3[1133] = {X 342.3291, Y 0.2255, Z -3.8333, A 0.000, B 0.000, C 0.000 }
gfCNCPoint3[1134] = {X 344.5718, Y -0.0335, Z -3.8333, A 0.000, B 0.000, C 0.000 }
gfCNCPoint3[1135] = {X 346.8284, Y -0.0996, Z -3.8333, A 0.000, B 0.000, C 0.000 }
gfCNCPoint3[1136] = {X 349.0824, Y 0.0276, Z -3.8333, A 0.000, B 0.000, C 0.000 }
gfCNCPoint3[1137] = {X 351.3172, Y 0.3472, Z -3.8333, A 0.000, B 0.000, C 0.000 }
gfCNCPoint3[1138] = {X 351.8877, Y 0.4533, Z -3.8333, A 0.000, B 0.000, C 0.000 }
gfCNCPoint3[1139] = {X 353.8296, Y 0.9413, Z -3.8333, A 0.000, B 0.000, C 0.000 }
gfCNCPoint3[1140] = {X 355.7165, Y 1.6111, Z -3.8333, A 0.000, B 0.000, C 0.000 }
gfCNCPoint3[1141] = {X 357.5314, Y 2.4567, Z -3.8333, A 0.000, B 0.000, C 0.000 }
gfCNCPoint3[1142] = {X 359.2580, Y 3.4705, Z -3.8333, A 0.000, B 0.000, C 0.000 }
gfCNCPoint3[1143] = {X 360.8807, Y 4.6434, Z -3.8333, A 0.000, B 0.000, C 0.000 }
gfCNCPoint3[1144] = {X 362.3850, Y 5.9648, Z -3.8333, A 0.000, B 0.000, C 0.000 }
gfCNCPoint3[1145] = {X 363.7572, Y 7.4229, Z -3.8333, A 0.000, B 0.000, C 0.000 }
gfCNCPoint3[1146] = {X 365.2278, Y 9.3208, Z -3.8333, A 0.000, B 0.000, C 0.000 }
gfCNCPoint3[1147] = {X 366.5080, Y 11.3520, Z -3.8333, A 0.000, B 0.000, C 0.000 }
gfCNCPoint3[1148] = {X 367.5857, Y 13.4974, Z -3.8333, A 0.000, B 0.000, C 0.000 }
gfCNCPoint3[1149] = {X 368.4508, Y 15.7371, Z -3.8333, A 0.000, B 0.000, C 0.000 }
gfCNCPoint3[1150] = {X 369.0954, Y 18.0499, Z -3.8333, A 0.000, B 0.000, C 0.000 }
gfCNCPoint3[1151] = {X 369.5789, Y 20.6929, Z -3.8333, A 0.000, B 0.000, C 0.000 }
gfCNCPoint3[1152] = {X 369.8369, Y 23.3674, Z -3.8333, A 0.000, B 0.000, C 0.000 }
gfCNCPoint3[1153] = {X 369.8675, Y 26.0541, Z -3.8333, A 0.000, B 0.000, C 0.000 }
gfCNCPoint3[1154] = {X 369.6704, Y 28.7338, Z -3.8333, A 0.000, B 0.000, C 0.000 }
gfCNCPoint3[1155] = {X 369.2471, Y 31.3871, Z -3.8333, A 0.000, B 0.000, C 0.000 }
gfCNCPoint3[1156] = {X 368.7215, Y 33.4981, Z -3.8333, A 0.000, B 0.000, C 0.000 }
gfCNCPoint3[1157] = {X 368.0115, Y 35.5545, Z -3.8333, A 0.000, B 0.000, C 0.000 }
gfCNCPoint3[1158] = {X 367.1226, Y 37.5401, Z -3.8333, A 0.000, B 0.000, C 0.000 }
gfCNCPoint3[1159] = {X 366.0618, Y 39.4394, Z -3.8333, A 0.000, B 0.000, C 0.000 }
gfCNCPoint3[1160] = {X 364.8373, Y 41.2375, Z -3.8333, A 0.000, B 0.000, C 0.000 }
gfCNCPoint3[1161] = {X 364.7112, Y 41.4096, Z -3.8333, A 0.000, B 0.000, C 0.000 }
gfCNCPoint3[1162] = {X 364.0852, Y 42.1781, Z -3.8333, A 0.000, B 0.000, C 0.000 }
gfCNCPoint3[1163] = {X 362.8197, Y 43.5979, Z -3.8333, A 0.000, B 0.000, C 0.000 }
gfCNCPoint3[1164] = {X 361.4329, Y 44.8996, Z -3.8333, A 0.000, B 0.000, C 0.000 }
gfCNCPoint3[1165] = {X 359.9359, Y 46.0729, Z -3.8333, A 0.000, B 0.000, C 0.000 }
gfCNCPoint3[1166] = {X 358.3405, Y 47.1085, Z -3.8333, A 0.000, B 0.000, C 0.000 }
gfCNCPoint3[1167] = {X 356.6594, Y 47.9981, Z -3.8333, A 0.000, B 0.000, C 0.000 }
gfCNCPoint3[1168] = {X 356.2500, Y 48.1918, Z -3.8333, A 0.000, B 0.000, C 0.000 }
gfCNCPoint3[1169] = {X 354.0457, Y 49.0143, Z -3.8333, A 0.000, B 0.000, C 0.000 }
gfCNCPoint3[1170] = {X 351.7691, Y 49.6083, Z -3.8333, A 0.000, B 0.000, C 0.000 }
gfCNCPoint3[1171] = {X 349.4440, Y 49.9677, Z -3.8333, A 0.000, B 0.000, C 0.000 }
gfCNCPoint3[1172] = {X 347.0943, Y 50.0886, Z -3.8333, A 0.000, B 0.000, C 0.000 }
gfCNCPoint3[1173] = {X 345.0202, Y 50.0535, Z -3.8333, A 0.000, B 0.000, C 0.000 }
gfCNCPoint3[1174] = {X 342.9569, Y 49.8386, Z -3.8333, A 0.000, B 0.000, C 0.000 }
gfCNCPoint3[1175] = {X 340.9201, Y 49.4455, Z -3.8333, A 0.000, B 0.000, C 0.000 }
gfCNCPoint3[1176] = {X 338.9250, Y 48.8771, Z -3.8333, A 0.000, B 0.000, C 0.000 }
gfCNCPoint3[1177] = {X 336.9868, Y 48.1378, Z -3.8333, A 0.000, B 0.000, C 0.000 }
gfCNCPoint3[1178] = {X 335.1200, Y 47.2332, Z -3.8333, A 0.000, B 0.000, C 0.000 }
gfCNCPoint3[1179] = {X 333.5417, Y 46.2595, Z -3.8333, A 0.000, B 0.000, C 0.000 }
gfCNCPoint3[1180] = {X 332.0435, Y 45.1663, Z -3.8333, A 0.000, B 0.000, C 0.000 }
gfCNCPoint3[1181] = {X 330.6346, Y 43.9603, Z -3.8333, A 0.000, B 0.000, C 0.000 }
gfCNCPoint3[1182] = {X 329.6760, Y 43.9518, Z -3.8333, A 0.000, B 0.000, C 0.000 }
gfCNCPoint3[1183] = {X 328.7421, Y 43.7359, Z -3.8333, A 0.000, B 0.000, C 0.000 }
gfCNCPoint3[1184] = {X 327.8770, Y 43.3228, Z -3.8333, A 0.000, B 0.000, C 0.000 }
gfCNCPoint3[1185] = {X 327.1219, Y 42.7321, Z -3.8333, A 0.000, B 0.000, C 0.000 }
gfCNCPoint3[1186] = {X 326.5249, Y 42.1498, Z -3.8333, A 0.000, B 0.000, C 0.000 }
gfCNCPoint3[1187] = {X 325.8848, Y 41.3619, Z -3.8333, A 0.000, B 0.000, C 0.000 }
gfCNCPoint3[1188] = {X 325.4424, Y 40.4483, Z -3.8333, A 0.000, B 0.000, C 0.000 }
gfCNCPoint3[1189] = {X 325.2210, Y 39.4576, Z -3.8333, A 0.000, B 0.000, C 0.000 }
gfCNCPoint3[1190] = {X 325.2326, Y 38.4426, Z -3.8333, A 0.000, B 0.000, C 0.000 }
gfCNCPoint3[1191] = {X 325.4765, Y 37.4572, Z -3.8333, A 0.000, B 0.000, C 0.000 }
gfCNCPoint3[1192] = {X 325.9397, Y 36.5539, Z -3.8333, A 0.000, B 0.000, C 0.000 }
gfCNCPoint3[1193] = {X 330.1988, Y 30.1861, Z -3.8333, A 0.000, B 0.000, C 0.000 }
gfCNCPoint3[1194] = {X 330.8195, Y 29.4619, Z -3.8333, A 0.000, B 0.000, C 0.000 }
gfCNCPoint3[1195] = {X 331.5816, Y 28.8884, Z -3.8333, A 0.000, B 0.000, C 0.000 }
gfCNCPoint3[1196] = {X 332.4495, Y 28.4927, Z -3.8333, A 0.000, B 0.000, C 0.000 }
gfCNCPoint3[1197] = {X 333.3822, Y 28.2932, Z -3.8333, A 0.000, B 0.000, C 0.000 }
gfCNCPoint3[1198] = {X 334.3360, Y 28.2995, Z -3.8333, A 0.000, B 0.000, C 0.000 }
gfCNCPoint3[1199] = {X 335.2660, Y 28.5111, Z -3.8333, A 0.000, B 0.000, C 0.000 }
gfCNCPoint3[1200] = {X 336.1286, Y 28.9182, Z -3.8333, A 0.000, B 0.000, C 0.000 }
gfCNCPoint3[1201] = {X 336.8832, Y 29.5016, Z -3.8333, A 0.000, B 0.000, C 0.000 }
gfCNCPoint3[1202] = {X 337.4845, Y 30.0811, Z -3.8333, A 0.000, B 0.000, C 0.000 }
gfCNCPoint3[1203] = {X 338.1273, Y 30.8804, Z -3.8333, A 0.000, B 0.000, C 0.000 }
gfCNCPoint3[1204] = {X 338.5677, Y 31.8067, Z -3.8333, A 0.000, B 0.000, C 0.000 }
gfCNCPoint3[1205] = {X 338.7817, Y 32.8098, Z -3.8333, A 0.000, B 0.000, C 0.000 }
gfCNCPoint3[1206] = {X 338.7576, Y 33.8352, Z -3.8333, A 0.000, B 0.000, C 0.000 }
gfCNCPoint3[1207] = {X 339.5037, Y 34.5088, Z -3.8333, A 0.000, B 0.000, C 0.000 }
gfCNCPoint3[1208] = {X 340.2822, Y 35.1446, Z -3.8333, A 0.000, B 0.000, C 0.000 }
gfCNCPoint3[1209] = {X 341.4935, Y 35.9468, Z -3.8333, A 0.000, B 0.000, C 0.000 }
gfCNCPoint3[1210] = {X 342.8036, Y 36.5748, Z -3.8333, A 0.000, B 0.000, C 0.000 }
gfCNCPoint3[1211] = {X 344.1877, Y 37.0165, Z -3.8333, A 0.000, B 0.000, C 0.000 }
gfCNCPoint3[1212] = {X 345.6193, Y 37.2636, Z -3.8333, A 0.000, B 0.000, C 0.000 }
gfCNCPoint3[1213] = {X 347.0713, Y 37.3115, Z -3.8333, A 0.000, B 0.000, C 0.000 }
gfCNCPoint3[1214] = {X 347.5139, Y 37.2886, Z -3.8333, A 0.000, B 0.000, C 0.000 }
gfCNCPoint3[1215] = {X 348.9409, Y 37.0970, Z -3.8333, A 0.000, B 0.000, C 0.000 }
gfCNCPoint3[1216] = {X 350.3177, Y 36.6757, Z -3.8333, A 0.000, B 0.000, C 0.000 }
gfCNCPoint3[1217] = {X 351.6076, Y 36.0358, Z -3.8333, A 0.000, B 0.000, C 0.000 }
gfCNCPoint3[1218] = {X 352.7761, Y 35.1946, Z -3.8333, A 0.000, B 0.000, C 0.000 }
gfCNCPoint3[1219] = {X 353.9225, Y 34.0810, Z -3.8333, A 0.000, B 0.000, C 0.000 }
gfCNCPoint3[1220] = {X 354.9147, Y 32.8281, Z -3.8333, A 0.000, B 0.000, C 0.000 }
gfCNCPoint3[1221] = {X 355.7358, Y 31.4569, Z -3.8333, A 0.000, B 0.000, C 0.000 }
gfCNCPoint3[1222] = {X 356.3719, Y 29.9907, Z -3.8333, A 0.000, B 0.000, C 0.000 }
gfCNCPoint3[1223] = {X 356.8123, Y 28.4543, Z -3.8333, A 0.000, B 0.000, C 0.000 }
